LIN {X 0,Y 623.912,Z 1169.845,A -85,B 0,C 180,E1 30061.655,E2 30061.655} C_VEL
LIN {X 0,Y 623.911,Z 1170.404,A -85,B 0,C 180,E1 30059.543,E2 30059.543} C_VEL
LIN {X 0,Y 623.904,Z 1169.363,A -85,B 0,C 180,E1 30057.614,E2 30057.614} C_VEL
LIN {X 0,Y 623.916,Z 1166.7,A -85,B 0,C 180,E1 30055.682,E2 30055.682} C_VEL
LIN {X 0,Y 623.959,Z 1162.568,A -85,B 0,C 180,E1 30053.746,E2 30053.746} C_VEL
LIN {X 0,Y 624.049,Z 1156.994,A -85,B 0,C 180,E1 30051.897,E2 30051.897} C_VEL
LIN {X 0,Y 624.248,Z 1149.09,A -85,B 0,C 180,E1 30049.854,E2 30049.854} C_VEL
LIN {X 0,Y 624.565,Z 1140.192,A -85,B 0,C 180,E1 30047.99,E2 30047.99} C_VEL
LIN {X 0,Y 625.015,Z 1129.706,A -85,B 0,C 180,E1 30046.186,E2 30046.186} C_VEL
LIN {X 0,Y 625.63,Z 1117.625,A -85,B 0,C 180,E1 30044.427,E2 30044.427} C_VEL
LIN {X 0,Y 626.415,Z 1103.895,A -85,B 0,C 180,E1 30042.731,E2 30042.731} C_VEL
LIN {X 0,Y 627.334,Z 1088.573,A -85,B 0,C 180,E1 30041.124,E2 30041.124} C_VEL
LIN {X 0,Y 628.363,Z 1072.134,A -85,B 0,C 180,E1 30039.656,E2 30039.656} C_VEL
LIN {X 0,Y 629.487,Z 1054.056,A -85,B 0,C 180,E1 30038.281,E2 30038.281} C_VEL
LIN {X 0,Y 630.63,Z 1034.884,A -85,B 0,C 180,E1 30037.045,E2 30037.045} C_VEL
LIN {X 0,Y 631.734,Z 1015.659,A -85,B 0,C 180,E1 30036.001,E2 30036.001} C_VEL
LIN {X 0,Y 632.769,Z 994.956,A -85,B 0,C 180,E1 30035.077,E2 30035.077} C_VEL
LIN {X 0,Y 633.68,Z 974.386,A -85,B 0,C 180,E1 30034.336,E2 30034.336} C_VEL
LIN {X 0,Y 634.446,Z 952.859,A -85,B 0,C 180,E1 30033.726,E2 30033.726} C_VEL
LIN {X 0,Y 635.069,Z 931.038,A -85,B 0,C 180,E1 30033.278,E2 30033.278} C_VEL
LIN {X 0,Y 635.631,Z 892.123,A -85,B 0,C 180,E1 30032.768,E2 30032.768} C_VEL
LIN {X 0,Y 637.752,Z 731.192,A -85,B 0,C 180,E1 30030.768,E2 30030.768} C_VEL
LIN {X 0,Y 637.014,Z 723.617,A -85,B 0,C 180,E1 30030.63,E2 30030.63} C_VEL
LIN {X 0,Y 631.874,Z 703.847,A -85,B 0,C 180,E1 30030.101,E2 30030.101} C_VEL
LIN {X 0,Y 631.316,Z 697.339,A -85,B 0,C 180,E1 30029.982,E2 30029.982} C_VEL
LIN {X 0,Y 631.888,Z 655.219,A -85,B 0,C 180,E1 30029.42,E2 30029.42} C_VEL
LIN {X 0,Y 618.767,Z 628.94,A -85,B 0,C 180,E1 30028.33,E2 30028.33} C_VEL
LIN {X 0,Y 617.781,Z 626.772,A -85,B 0,C 180,E1 30028.226,E2 30028.226} C_VEL
LIN {X 0,Y 616.937,Z 623.823,A -85,B 0,C 180,E1 30027.835,E2 30027.835} C_VEL
LIN {X 0,Y 617.007,Z 623.813,A -85,B 0,C 180,E1 30024.762,E2 30024.762} C_VEL
LIN {X 0,Y 616.975,Z 623.812,A -85,B 0,C 180,E1 30021.636,E2 30021.636} C_VEL
LIN {X 0,Y 617.012,Z 623.805,A -85,B 0,C 180,E1 30018.478,E2 30018.478} C_VEL
LIN {X 0,Y 616.987,Z 623.813,A -85,B 0,C 180,E1 30015.221,E2 30015.221} C_VEL
LIN {X 0,Y 617.016,Z 623.81,A -85,B 0,C 180,E1 30012.085,E2 30012.085} C_VEL
LIN {X 0,Y 616.929,Z 623.818,A -85,B 0,C 180,E1 30009.078,E2 30009.078} C_VEL
LIN {X 0,Y 617.013,Z 623.809,A -85,B 0,C 180,E1 30006.034,E2 30006.034} C_VEL
LIN {X 0,Y 616.994,Z 623.814,A -85,B 0,C 180,E1 30002.882,E2 30002.882} C_VEL
LIN {X 0,Y 617.01,Z 623.806,A -85,B 0,C 180,E1 29999.622,E2 29999.622} C_VEL
LIN {X 0,Y 616.974,Z 623.811,A -85,B 0,C 180,E1 29996.551,E2 29996.551} C_VEL
LIN {X 0,Y 617.005,Z 623.814,A -85,B 0,C 180,E1 29993.394,E2 29993.394} C_VEL
LIN {X 0,Y 616.935,Z 623.817,A -85,B 0,C 180,E1 29990.394,E2 29990.394} C_VEL
LIN {X 0,Y 616.989,Z 623.809,A -85,B 0,C 180,E1 29987.253,E2 29987.253} C_VEL
LIN {X 0,Y 617.016,Z 623.808,A -85,B 0,C 180,E1 29984.165,E2 29984.165} C_VEL
LIN {X 0,Y 617.008,Z 623.81,A -85,B 0,C 180,E1 29980.889,E2 29980.889} C_VEL
LIN {X 0,Y 616.968,Z 623.808,A -85,B 0,C 180,E1 29977.825,E2 29977.825} C_VEL
LIN {X 0,Y 616.969,Z 623.815,A -85,B 0,C 180,E1 29974.697,E2 29974.697} C_VEL
LIN {X 0,Y 616.953,Z 623.81,A -85,B 0,C 180,E1 29971.673,E2 29971.673} C_VEL
LIN {X 0,Y 616.975,Z 623.81,A -85,B 0,C 180,E1 29968.515,E2 29968.515} C_VEL
LIN {X 0,Y 617.007,Z 623.807,A -85,B 0,C 180,E1 29965.447,E2 29965.447} C_VEL
LIN {X 0,Y 617.012,Z 623.811,A -85,B 0,C 180,E1 29962.271,E2 29962.271} C_VEL
LIN {X 0,Y 616.964,Z 623.804,A -85,B 0,C 180,E1 29959.26,E2 29959.26} C_VEL
LIN {X 0,Y 616.947,Z 623.816,A -85,B 0,C 180,E1 29956.027,E2 29956.027} C_VEL
LIN {X 0,Y 616.966,Z 623.815,A -85,B 0,C 180,E1 29953.138,E2 29953.138} C_VEL
LIN {X 0,Y 616.98,Z 623.809,A -85,B 0,C 180,E1 29950.006,E2 29950.006} C_VEL
LIN {X 0,Y 617.004,Z 623.809,A -85,B 0,C 180,E1 29946.912,E2 29946.912} C_VEL
LIN {X 0,Y 617.013,Z 623.812,A -85,B 0,C 180,E1 29943.744,E2 29943.744} C_VEL
LIN {X 0,Y 616.963,Z 623.813,A -85,B 0,C 180,E1 29940.698,E2 29940.698} C_VEL
LIN {X 0,Y 616.938,Z 623.817,A -85,B 0,C 180,E1 29937.429,E2 29937.429} C_VEL
LIN {X 0,Y 616.985,Z 623.816,A -85,B 0,C 180,E1 29934.539,E2 29934.539} C_VEL
LIN {X 0,Y 616.98,Z 623.811,A -85,B 0,C 180,E1 29931.36,E2 29931.36} C_VEL
LIN {X 0,Y 617,Z 623.81,A -85,B 0,C 180,E1 29928.334,E2 29928.334} C_VEL
LIN {X 0,Y 617.01,Z 623.811,A -85,B 0,C 180,E1 29925.179,E2 29925.179} C_VEL
LIN {X 0,Y 616.963,Z 623.816,A -85,B 0,C 180,E1 29922.137,E2 29922.137} C_VEL
LIN {X 0,Y 616.934,Z 623.827,A -85,B 0,C 180,E1 29920.696,E2 29920.696} C_VEL
LIN {X 0,Y 622.527,Z 645.232,A -85,B 0,C 180,E1 29918.834,E2 29918.834} C_VEL
LIN {X 0,Y 621.851,Z 690.99,A -85,B 0,C 180,E1 29915.395,E2 29915.395} C_VEL
LIN {X 0,Y 621.209,Z 730.49,A -85,B 0,C 180,E1 29912.408,E2 29912.408} C_VEL
LIN {X 0,Y 620.43,Z 772.737,A -85,B 0,C 180,E1 29909.227,E2 29909.227} C_VEL
LIN {X 0,Y 619.705,Z 815.192,A -85,B 0,C 180,E1 29906.029,E2 29906.029} C_VEL
LIN {X 0,Y 619.607,Z 824.743,A -85,B 0,C 180,E1 29905.342,E2 29905.342} C_VEL
LIN {X 0,Y 619.958,Z 832.218,A -85,B 0,C 180,E1 29905.238,E2 29905.238} C_VEL
LIN {X 0,Y 618.985,Z 967.136,A -85,B 0,C 180,E1 29903.544,E2 29903.544} C_VEL
LIN {X 0,Y 618.854,Z 983.402,A -85,B 0,C 180,E1 29903.165,E2 29903.165} C_VEL
LIN {X 0,Y 618.641,Z 999.258,A -85,B 0,C 180,E1 29902.621,E2 29902.621} C_VEL
LIN {X 0,Y 618.348,Z 1013.981,A -85,B 0,C 180,E1 29901.931,E2 29901.931} C_VEL
LIN {X 0,Y 618.043,Z 1027.886,A -85,B 0,C 180,E1 29901.096,E2 29901.096} C_VEL
LIN {X 0,Y 617.697,Z 1040.445,A -85,B 0,C 180,E1 29900.144,E2 29900.144} C_VEL
LIN {X 0,Y 617.356,Z 1052.594,A -85,B 0,C 180,E1 29898.996,E2 29898.996} C_VEL
LIN {X 0,Y 617.064,Z 1062.411,A -85,B 0,C 180,E1 29897.831,E2 29897.831} C_VEL
LIN {X 0,Y 616.819,Z 1071.471,A -85,B 0,C 180,E1 29896.478,E2 29896.478} C_VEL
LIN {X 0,Y 616.646,Z 1078.364,A -85,B 0,C 180,E1 29895.131,E2 29895.131} C_VEL
LIN {X 0,Y 616.54,Z 1083.784,A -85,B 0,C 180,E1 29893.694,E2 29893.694} C_VEL
LIN {X 0,Y 616.468,Z 1087.777,A -85,B 0,C 180,E1 29892.039,E2 29892.039} C_VEL
LIN {X 0,Y 616.45,Z 1089.511,A -85,B 0,C 180,E1 29890.559,E2 29890.559} C_VEL
LIN {X 0,Y 616.474,Z 1089.436,A -85,B 0,C 180,E1 29889.05,E2 29889.05} C_VEL
LIN {X 0,Y 616.534,Z 1087.628,A -85,B 0,C 180,E1 29887.546,E2 29887.546} C_VEL
LIN {X 0,Y 616.626,Z 1083.923,A -85,B 0,C 180,E1 29886.048,E2 29886.048} C_VEL
LIN {X 0,Y 616.778,Z 1078.713,A -85,B 0,C 180,E1 29884.647,E2 29884.647} C_VEL
LIN {X 0,Y 616.991,Z 1071.524,A -85,B 0,C 180,E1 29883.25,E2 29883.25} C_VEL
LIN {X 0,Y 617.267,Z 1062.829,A -85,B 0,C 180,E1 29881.947,E2 29881.947} C_VEL
LIN {X 0,Y 617.594,Z 1052.516,A -85,B 0,C 180,E1 29880.74,E2 29880.74} C_VEL
LIN {X 0,Y 617.96,Z 1040.631,A -85,B 0,C 180,E1 29879.627,E2 29879.627} C_VEL
LIN {X 0,Y 618.306,Z 1027.459,A -85,B 0,C 180,E1 29878.654,E2 29878.654} C_VEL
LIN {X 0,Y 618.576,Z 1014.097,A -85,B 0,C 180,E1 29877.867,E2 29877.867} C_VEL
LIN {X 0,Y 618.83,Z 999.677,A -85,B 0,C 180,E1 29877.22,E2 29877.22} C_VEL
LIN {X 0,Y 619.005,Z 985.719,A -85,B 0,C 180,E1 29876.748,E2 29876.748} C_VEL
LIN {X 0,Y 619.098,Z 970.478,A -85,B 0,C 180,E1 29876.378,E2 29876.378} C_VEL
LIN {X 0,Y 619.279,Z 928.275,A -85,B 0,C 180,E1 29875.826,E2 29875.826} C_VEL
LIN {X 0,Y 620.272,Z 827.99,A -85,B 0,C 180,E1 29874.517,E2 29874.517} C_VEL
LIN {X 0,Y 620.921,Z 785.093,A -85,B 0,C 180,E1 29871.338,E2 29871.338} C_VEL
LIN {X 0,Y 621.362,Z 749.405,A -85,B 0,C 180,E1 29868.723,E2 29868.723} C_VEL
LIN {X 0,Y 621.787,Z 707.503,A -85,B 0,C 180,E1 29865.708,E2 29865.708} C_VEL
LIN {X 0,Y 621.849,Z 662.544,A -85,B 0,C 180,E1 29862.548,E2 29862.548} C_VEL
LIN {X 0,Y 621.705,Z 640.309,A -85,B 0,C 180,E1 29861.022,E2 29861.022} C_VEL
LIN {X 0,Y 616.991,Z 623.817,A -85,B 0,C 180,E1 29859.681,E2 29859.681} C_VEL
LIN {X 0,Y 616.981,Z 623.82,A -85,B 0,C 180,E1 29856.706,E2 29856.706} C_VEL
LIN {X 0,Y 617.01,Z 623.814,A -85,B 0,C 180,E1 29853.326,E2 29853.326} C_VEL
LIN {X 0,Y 617.018,Z 623.814,A -85,B 0,C 180,E1 29850.105,E2 29850.105} C_VEL
LIN {X 0,Y 616.973,Z 623.815,A -85,B 0,C 180,E1 29846.895,E2 29846.895} C_VEL
LIN {X 0,Y 616.987,Z 623.814,A -85,B 0,C 180,E1 29843.963,E2 29843.963} C_VEL
LIN {X 0,Y 617.01,Z 623.814,A -85,B 0,C 180,E1 29840.68,E2 29840.68} C_VEL
LIN {X 0,Y 617.019,Z 623.81,A -85,B 0,C 180,E1 29837.486,E2 29837.486} C_VEL
LIN {X 0,Y 616.973,Z 623.813,A -85,B 0,C 180,E1 29834.247,E2 29834.247} C_VEL
LIN {X 0,Y 617.021,Z 623.809,A -85,B 0,C 180,E1 29831.016,E2 29831.016} C_VEL
LIN {X 0,Y 617.006,Z 623.811,A -85,B 0,C 180,E1 29827.887,E2 29827.887} C_VEL
LIN {X 0,Y 617.049,Z 624.04,A -85,B 0,C 180,E1 29826.952,E2 29826.952} C_VEL
LIN {X 0,Y 624.996,Z 648.862,A -85,B 0,C 180,E1 29824.16,E2 29824.16} C_VEL
LIN {X 0,Y 627.248,Z 656.87,A -85,B 0,C 180,E1 29823.308,E2 29823.308} C_VEL
LIN {X 0,Y 626.069,Z 680.989,A -85,B 0,C 180,E1 29821.26,E2 29821.26} C_VEL
LIN {X 0,Y 631.821,Z 709.359,A -85,B 0,C 180,E1 29820.55,E2 29820.55} C_VEL
LIN {X 0,Y 628.74,Z 911.351,A -85,B 0,C 180,E1 29817.97,E2 29817.97} C_VEL
LIN {X 0,Y 627.625,Z 986.56,A -85,B 0,C 180,E1 29816.998,E2 29816.998} C_VEL
LIN {X 0,Y 626.902,Z 1008.567,A -85,B 0,C 180,E1 29816.549,E2 29816.549} C_VEL
LIN {X 0,Y 626.04,Z 1030.132,A -85,B 0,C 180,E1 29815.944,E2 29815.944} C_VEL
LIN {X 0,Y 625.036,Z 1051.381,A -85,B 0,C 180,E1 29815.182,E2 29815.182} C_VEL
LIN {X 0,Y 623.929,Z 1072.004,A -85,B 0,C 180,E1 29814.265,E2 29814.265} C_VEL
LIN {X 0,Y 622.789,Z 1091.493,A -85,B 0,C 180,E1 29813.212,E2 29813.212} C_VEL
LIN {X 0,Y 621.585,Z 1111.078,A -85,B 0,C 180,E1 29811.961,E2 29811.961} C_VEL
LIN {X 0,Y 620.498,Z 1128.452,A -85,B 0,C 180,E1 29810.663,E2 29810.663} C_VEL
LIN {X 0,Y 619.474,Z 1144.894,A -85,B 0,C 180,E1 29809.22,E2 29809.22} C_VEL
LIN {X 0,Y 618.568,Z 1159.94,A -85,B 0,C 180,E1 29807.69,E2 29807.69} C_VEL
LIN {X 0,Y 617.799,Z 1173.773,A -85,B 0,C 180,E1 29806.065,E2 29806.065} C_VEL
LIN {X 0,Y 617.156,Z 1186.266,A -85,B 0,C 180,E1 29804.334,E2 29804.334} C_VEL
LIN {X 0,Y 616.677,Z 1197.217,A -85,B 0,C 180,E1 29802.547,E2 29802.547} C_VEL
LIN {X 0,Y 616.353,Z 1206.523,A -85,B 0,C 180,E1 29800.751,E2 29800.751} C_VEL
LIN {X 0,Y 616.121,Z 1214.386,A -85,B 0,C 180,E1 29798.867,E2 29798.867} C_VEL
LIN {X 0,Y 615.98,Z 1220.89,A -85,B 0,C 180,E1 29796.898,E2 29796.898} C_VEL
LIN {X 0,Y 615.92,Z 1225.641,A -85,B 0,C 180,E1 29794.935,E2 29794.935} C_VEL
LIN {X 0,Y 615.904,Z 1228.673,A -85,B 0,C 180,E1 29792.977,E2 29792.977} C_VEL
LIN {X 0,Y 615.91,Z 1230.28,A -85,B 0,C 180,E1 29790.929,E2 29790.929} C_VEL
LIN {X 0,Y 615.91,Z 1230.279,A -85,B 0,C 180,E1 29789.069,E2 29789.069} C_VEL
LIN {X 0,Y 615.905,Z 1228.666,A -85,B 0,C 180,E1 29787.021,E2 29787.021} C_VEL
LIN {X 0,Y 615.92,Z 1225.63,A -85,B 0,C 180,E1 29785.063,E2 29785.063} C_VEL
LIN {X 0,Y 615.981,Z 1220.882,A -85,B 0,C 180,E1 29783.1,E2 29783.1} C_VEL
LIN {X 0,Y 616.119,Z 1214.356,A -85,B 0,C 180,E1 29781.13,E2 29781.13} C_VEL
LIN {X 0,Y 616.35,Z 1206.432,A -85,B 0,C 180,E1 29779.247,E2 29779.247} C_VEL
LIN {X 0,Y 616.699,Z 1196.523,A -85,B 0,C 180,E1 29777.355,E2 29777.355} C_VEL
LIN {X 0,Y 617.182,Z 1185.19,A -85,B 0,C 180,E1 29775.551,E2 29775.551} C_VEL
LIN {X 0,Y 617.807,Z 1172.49,A -85,B 0,C 180,E1 29773.836,E2 29773.836} C_VEL
LIN {X 0,Y 618.569,Z 1158.134,A -85,B 0,C 180,E1 29772.196,E2 29772.196} C_VEL
LIN {X 0,Y 619.47,Z 1142.089,A -85,B 0,C 180,E1 29770.627,E2 29770.627} C_VEL
LIN {X 0,Y 620.503,Z 1124.219,A -85,B 0,C 180,E1 29769.137,E2 29769.137} C_VEL
LIN {X 0,Y 621.53,Z 1105.923,A -85,B 0,C 180,E1 29767.835,E2 29767.835} C_VEL
LIN {X 0,Y 622.596,Z 1086.571,A -85,B 0,C 180,E1 29766.678,E2 29766.678} C_VEL
LIN {X 0,Y 623.608,Z 1066.417,A -85,B 0,C 180,E1 29765.664,E2 29765.664} C_VEL
LIN {X 0,Y 624.581,Z 1045.558,A -85,B 0,C 180,E1 29764.795,E2 29764.795} C_VEL
LIN {X 0,Y 625.479,Z 1023.937,A -85,B 0,C 180,E1 29764.073,E2 29764.073} C_VEL
LIN {X 0,Y 626.217,Z 1002.185,A -85,B 0,C 180,E1 29763.519,E2 29763.519} C_VEL
LIN {X 0,Y 626.845,Z 978.254,A -85,B 0,C 180,E1 29763.087,E2 29763.087} C_VEL
LIN {X 0,Y 628.923,Z 830.62,A -85,B 0,C 180,E1 29761.18,E2 29761.18} C_VEL
LIN {X 0,Y 631.767,Z 708.547,A -85,B 0,C 180,E1 29759.452,E2 29759.452} C_VEL
LIN {X 0,Y 625.568,Z 675.462,A -85,B 0,C 180,E1 29758.5,E2 29758.5} C_VEL
LIN {X 0,Y 626.748,Z 655.477,A -85,B 0,C 180,E1 29756.714,E2 29756.714} C_VEL
LIN {X 0,Y 622.75,Z 640.651,A -85,B 0,C 180,E1 29754.972,E2 29754.972} C_VEL
LIN {X 0,Y 619,Z 629.633,A -85,B 0,C 180,E1 29753.487,E2 29753.487} C_VEL
LIN {X 0,Y 617.009,Z 623.813,A -85,B 0,C 180,E1 29752.602,E2 29752.602} C_VEL
LIN {X 0,Y 616.98,Z 623.818,A -85,B 0,C 180,E1 29749.59,E2 29749.59} C_VEL
LIN {X 0,Y 617.013,Z 623.813,A -85,B 0,C 180,E1 29746.47,E2 29746.47} C_VEL
LIN {X 0,Y 616.971,Z 623.817,A -85,B 0,C 180,E1 29743.407,E2 29743.407} C_VEL
LIN {X 0,Y 617.018,Z 623.813,A -85,B 0,C 180,E1 29740.286,E2 29740.286} C_VEL
LIN {X 0,Y 616.963,Z 623.817,A -85,B 0,C 180,E1 29737.273,E2 29737.273} C_VEL
LIN {X 0,Y 617.019,Z 623.812,A -85,B 0,C 180,E1 29734.218,E2 29734.218} C_VEL
LIN {X 0,Y 616.979,Z 623.96,A -85,B 0,C 180,E1 29733.382,E2 29733.382} C_VEL
LIN {X 0,Y 620.268,Z 633.467,A -85,B 0,C 180,E1 29731.798,E2 29731.798} C_VEL
LIN {X 0,Y 628.034,Z 646.969,A -85,B 0,C 180,E1 29731.002,E2 29731.002} C_VEL
LIN {X 0,Y 632.541,Z 656.333,A -85,B 0,C 180,E1 29730.544,E2 29730.544} C_VEL
LIN {X 0,Y 629.48,Z 777.376,A -85,B 0,C 180,E1 29728.801,E2 29728.801} C_VEL
LIN {X 0,Y 627.398,Z 908.624,A -85,B 0,C 180,E1 29727.084,E2 29727.084} C_VEL
LIN {X 0,Y 626.891,Z 937.237,A -85,B 0,C 180,E1 29726.668,E2 29726.668} C_VEL
LIN {X 0,Y 626.321,Z 959.429,A -85,B 0,C 180,E1 29726.177,E2 29726.177} C_VEL
LIN {X 0,Y 625.546,Z 980.68,A -85,B 0,C 180,E1 29725.544,E2 29725.544} C_VEL
LIN {X 0,Y 624.643,Z 1001.442,A -85,B 0,C 180,E1 29724.747,E2 29724.747} C_VEL
LIN {X 0,Y 623.606,Z 1021.962,A -85,B 0,C 180,E1 29723.783,E2 29723.783} C_VEL
LIN {X 0,Y 622.581,Z 1040.772,A -85,B 0,C 180,E1 29722.723,E2 29722.723} C_VEL
LIN {X 0,Y 621.481,Z 1058.677,A -85,B 0,C 180,E1 29721.522,E2 29721.522} C_VEL
LIN {X 0,Y 620.415,Z 1075.722,A -85,B 0,C 180,E1 29720.177,E2 29720.177} C_VEL
LIN {X 0,Y 619.416,Z 1091.38,A -85,B 0,C 180,E1 29718.739,E2 29718.739} C_VEL
LIN {X 0,Y 618.483,Z 1106.471,A -85,B 0,C 180,E1 29717.113,E2 29717.113} C_VEL
LIN {X 0,Y 617.681,Z 1119.911,A -85,B 0,C 180,E1 29715.397,E2 29715.397} C_VEL
LIN {X 0,Y 617.043,Z 1131.871,A -85,B 0,C 180,E1 29713.591,E2 29713.591} C_VEL
LIN {X 0,Y 616.563,Z 1142.344,A -85,B 0,C 180,E1 29711.698,E2 29711.698} C_VEL
LIN {X 0,Y 616.255,Z 1150.933,A -85,B 0,C 180,E1 29709.811,E2 29709.811} C_VEL
LIN {X 0,Y 616.053,Z 1158.018,A -85,B 0,C 180,E1 29707.838,E2 29707.838} C_VEL
LIN {X 0,Y 615.948,Z 1163.903,A -85,B 0,C 180,E1 29705.669,E2 29705.669} C_VEL
LIN {X 0,Y 615.915,Z 1167.665,A -85,B 0,C 180,E1 29703.725,E2 29703.725} C_VEL
LIN {X 0,Y 615.91,Z 1169.775,A -85,B 0,C 180,E1 29701.77,E2 29701.77} C_VEL
LIN {X 0,Y 615.905,Z 1170.449,A -85,B 0,C 180,E1 29699.723,E2 29699.723} C_VEL
LIN {X 0,Y 615.902,Z 1169.569,A -85,B 0,C 180,E1 29697.862,E2 29697.862} C_VEL
LIN {X 0,Y 615.91,Z 1167.023,A -85,B 0,C 180,E1 29695.813,E2 29695.813} C_VEL
LIN {X 0,Y 615.947,Z 1163.241,A -85,B 0,C 180,E1 29693.945,E2 29693.945} C_VEL
LIN {X 0,Y 616.051,Z 1157.696,A -85,B 0,C 180,E1 29691.978,E2 29691.978} C_VEL
LIN {X 0,Y 616.26,Z 1150.491,A -85,B 0,C 180,E1 29690.005,E2 29690.005} C_VEL
LIN {X 0,Y 616.58,Z 1141.807,A -85,B 0,C 180,E1 29688.117,E2 29688.117} C_VEL
LIN {X 0,Y 617.064,Z 1131.192,A -85,B 0,C 180,E1 29686.222,E2 29686.222} C_VEL
LIN {X 0,Y 617.723,Z 1118.936,A -85,B 0,C 180,E1 29684.39,E2 29684.39} C_VEL
LIN {X 0,Y 618.531,Z 1105.593,A -85,B 0,C 180,E1 29682.698,E2 29682.698} C_VEL
LIN {X 0,Y 619.497,Z 1090.283,A -85,B 0,C 180,E1 29681.055,E2 29681.055} C_VEL
LIN {X 0,Y 620.598,Z 1073.703,A -85,B 0,C 180,E1 29679.538,E2 29679.538} C_VEL
LIN {X 0,Y 621.774,Z 1055.841,A -85,B 0,C 180,E1 29678.146,E2 29678.146} C_VEL
LIN {X 0,Y 622.937,Z 1037.8,A -85,B 0,C 180,E1 29676.946,E2 29676.946} C_VEL
LIN {X 0,Y 624.116,Z 1018.173,A -85,B 0,C 180,E1 29675.849,E2 29675.849} C_VEL
LIN {X 0,Y 625.187,Z 998.226,A -85,B 0,C 180,E1 29674.926,E2 29674.926} C_VEL
LIN {X 0,Y 626.198,Z 977.222,A -85,B 0,C 180,E1 29674.134,E2 29674.134} C_VEL
LIN {X 0,Y 627.058,Z 955.646,A -85,B 0,C 180,E1 29673.494,E2 29673.494} C_VEL
LIN {X 0,Y 627.691,Z 933.727,A -85,B 0,C 180,E1 29673.025,E2 29673.025} C_VEL
LIN {X 0,Y 628.228,Z 904.066,A -85,B 0,C 180,E1 29672.608,E2 29672.608} C_VEL
LIN {X 0,Y 631.316,Z 697.339,A -85,B 0,C 180,E1 29669.982,E2 29669.982} C_VEL
LIN {X 0,Y 630.577,Z 689.773,A -85,B 0,C 180,E1 29669.838,E2 29669.838} C_VEL
LIN {X 0,Y 625.54,Z 670.016,A -85,B 0,C 180,E1 29669.294,E2 29669.294} C_VEL
LIN {X 0,Y 624.995,Z 663.512,A -85,B 0,C 180,E1 29669.173,E2 29669.173} C_VEL
LIN {X 0,Y 624.879,Z 657.552,A -85,B 0,C 180,E1 29669.081,E2 29669.081} C_VEL
LIN {X 0,Y 611.174,Z 630.338,A -85,B 0,C 180,E1 29667.915,E2 29667.915} C_VEL
LIN {X 0,Y 609.654,Z 627.14,A -85,B 0,C 180,E1 29667.767,E2 29667.767} C_VEL
LIN {X 0,Y 608.993,Z 624.813,A -85,B 0,C 180,E1 29667.447,E2 29667.447} C_VEL
LIN {X 0,Y 609.041,Z 624.803,A -85,B 0,C 180,E1 29664.239,E2 29664.239} C_VEL
LIN {X 0,Y 609.069,Z 624.803,A -85,B 0,C 180,E1 29661.166,E2 29661.166} C_VEL
LIN {X 0,Y 609.062,Z 624.797,A -85,B 0,C 180,E1 29657.907,E2 29657.907} C_VEL
LIN {X 0,Y 609.038,Z 624.8,A -85,B 0,C 180,E1 29654.831,E2 29654.831} C_VEL
LIN {X 0,Y 609.043,Z 624.806,A -85,B 0,C 180,E1 29651.674,E2 29651.674} C_VEL
LIN {X 0,Y 609.004,Z 624.807,A -85,B 0,C 180,E1 29648.723,E2 29648.723} C_VEL
LIN {X 0,Y 609.029,Z 624.799,A -85,B 0,C 180,E1 29645.485,E2 29645.485} C_VEL
LIN {X 0,Y 609.074,Z 624.8,A -85,B 0,C 180,E1 29642.461,E2 29642.461} C_VEL
LIN {X 0,Y 609.068,Z 624.799,A -85,B 0,C 180,E1 29639.29,E2 29639.29} C_VEL
LIN {X 0,Y 609.038,Z 624.798,A -85,B 0,C 180,E1 29636.209,E2 29636.209} C_VEL
LIN {X 0,Y 609.01,Z 624.803,A -85,B 0,C 180,E1 29632.926,E2 29632.926} C_VEL
LIN {X 0,Y 609.032,Z 624.806,A -85,B 0,C 180,E1 29629.969,E2 29629.969} C_VEL
LIN {X 0,Y 609.028,Z 624.8,A -85,B 0,C 180,E1 29626.796,E2 29626.796} C_VEL
LIN {X 0,Y 609.067,Z 624.793,A -85,B 0,C 180,E1 29623.772,E2 29623.772} C_VEL
LIN {X 0,Y 609.07,Z 624.803,A -85,B 0,C 180,E1 29620.501,E2 29620.501} C_VEL
LIN {X 0,Y 609.056,Z 624.795,A -85,B 0,C 180,E1 29617.358,E2 29617.358} C_VEL
LIN {X 0,Y 608.994,Z 624.803,A -85,B 0,C 180,E1 29614.238,E2 29614.238} C_VEL
LIN {X 0,Y 609.076,Z 624.801,A -85,B 0,C 180,E1 29611.13,E2 29611.13} C_VEL
LIN {X 0,Y 609.036,Z 624.801,A -85,B 0,C 180,E1 29608.026,E2 29608.026} C_VEL
LIN {X 0,Y 609.072,Z 624.79,A -85,B 0,C 180,E1 29604.821,E2 29604.821} C_VEL
LIN {X 0,Y 609.044,Z 624.799,A -85,B 0,C 180,E1 29601.6,E2 29601.6} C_VEL
LIN {X 0,Y 609.074,Z 624.791,A -85,B 0,C 180,E1 29598.448,E2 29598.448} C_VEL
LIN {X 0,Y 608.989,Z 624.805,A -85,B 0,C 180,E1 29595.453,E2 29595.453} C_VEL
LIN {X 0,Y 609.05,Z 624.799,A -85,B 0,C 180,E1 29592.321,E2 29592.321} C_VEL
LIN {X 0,Y 609.064,Z 624.802,A -85,B 0,C 180,E1 29589.233,E2 29589.233} C_VEL
LIN {X 0,Y 609.066,Z 624.796,A -85,B 0,C 180,E1 29585.977,E2 29585.977} C_VEL
LIN {X 0,Y 609.038,Z 624.8,A -85,B 0,C 180,E1 29582.952,E2 29582.952} C_VEL
LIN {X 0,Y 609.062,Z 624.804,A -85,B 0,C 180,E1 29579.846,E2 29579.846} C_VEL
LIN {X 0,Y 608.997,Z 624.806,A -85,B 0,C 180,E1 29576.856,E2 29576.856} C_VEL
LIN {X 0,Y 609.033,Z 624.8,A -85,B 0,C 180,E1 29573.553,E2 29573.553} C_VEL
LIN {X 0,Y 609.074,Z 624.802,A -85,B 0,C 180,E1 29570.491,E2 29570.491} C_VEL
LIN {X 0,Y 609.068,Z 624.8,A -85,B 0,C 180,E1 29567.314,E2 29567.314} C_VEL
LIN {X 0,Y 609.036,Z 624.802,A -85,B 0,C 180,E1 29564.242,E2 29564.242} C_VEL
LIN {X 0,Y 609.015,Z 624.843,A -85,B 0,C 180,E1 29560.957,E2 29560.957} C_VEL
LIN {X 0,Y 614.93,Z 647.129,A -85,B 0,C 180,E1 29558.993,E2 29558.993} C_VEL
LIN {X 0,Y 614.222,Z 691.425,A -85,B 0,C 180,E1 29555.643,E2 29555.643} C_VEL
LIN {X 0,Y 613.557,Z 731.688,A -85,B 0,C 180,E1 29552.595,E2 29552.595} C_VEL
LIN {X 0,Y 612.717,Z 774.101,A -85,B 0,C 180,E1 29549.379,E2 29549.379} C_VEL
LIN {X 0,Y 611.96,Z 816.445,A -85,B 0,C 180,E1 29546.175,E2 29546.175} C_VEL
LIN {X 0,Y 611.854,Z 825.417,A -85,B 0,C 180,E1 29545.524,E2 29545.524} C_VEL
LIN {X 0,Y 612.206,Z 832.974,A -85,B 0,C 180,E1 29545.416,E2 29545.416} C_VEL
LIN {X 0,Y 611.162,Z 968.04,A -85,B 0,C 180,E1 29543.688,E2 29543.688} C_VEL
LIN {X 0,Y 611.028,Z 984.393,A -85,B 0,C 180,E1 29543.3,E2 29543.3} C_VEL
LIN {X 0,Y 610.815,Z 999.568,A -85,B 0,C 180,E1 29542.774,E2 29542.774} C_VEL
LIN {X 0,Y 610.511,Z 1014.46,A -85,B 0,C 180,E1 29542.076,E2 29542.076} C_VEL
LIN {X 0,Y 610.177,Z 1029.016,A -85,B 0,C 180,E1 29541.192,E2 29541.192} C_VEL
LIN {X 0,Y 609.805,Z 1041.758,A -85,B 0,C 180,E1 29540.208,E2 29540.208} C_VEL
LIN {X 0,Y 609.454,Z 1053.779,A -85,B 0,C 180,E1 29539.053,E2 29539.053} C_VEL
LIN {X 0,Y 609.123,Z 1064.262,A -85,B 0,C 180,E1 29537.775,E2 29537.775} C_VEL
LIN {X 0,Y 608.884,Z 1072.789,A -85,B 0,C 180,E1 29536.466,E2 29536.466} C_VEL
LIN {X 0,Y 608.695,Z 1079.955,A -85,B 0,C 180,E1 29535.016,E2 29535.016} C_VEL
LIN {X 0,Y 608.594,Z 1085.137,A -85,B 0,C 180,E1 29533.586,E2 29533.586} C_VEL
LIN {X 0,Y 608.519,Z 1088.89,A -85,B 0,C 180,E1 29531.946,E2 29531.946} C_VEL
LIN {X 0,Y 608.505,Z 1090.475,A -85,B 0,C 180,E1 29530.507,E2 29530.507} C_VEL
LIN {X 0,Y 608.535,Z 1090.359,A -85,B 0,C 180,E1 29528.978,E2 29528.978} C_VEL
LIN {X 0,Y 608.602,Z 1088.497,A -85,B 0,C 180,E1 29527.455,E2 29527.455} C_VEL
LIN {X 0,Y 608.709,Z 1084.728,A -85,B 0,C 180,E1 29525.938,E2 29525.938} C_VEL
LIN {X 0,Y 608.881,Z 1079.447,A -85,B 0,C 180,E1 29524.519,E2 29524.519} C_VEL
LIN {X 0,Y 609.115,Z 1072.156,A -85,B 0,C 180,E1 29523.103,E2 29523.103} C_VEL
LIN {X 0,Y 609.415,Z 1063.348,A -85,B 0,C 180,E1 29521.784,E2 29521.784} C_VEL
LIN {X 0,Y 609.771,Z 1052.896,A -85,B 0,C 180,E1 29520.562,E2 29520.562} C_VEL
LIN {X 0,Y 610.146,Z 1041.389,A -85,B 0,C 180,E1 29519.482,E2 29519.482} C_VEL
LIN {X 0,Y 610.516,Z 1028.178,A -85,B 0,C 180,E1 29518.496,E2 29518.496} C_VEL
LIN {X 0,Y 610.807,Z 1014.75,A -85,B 0,C 180,E1 29517.699,E2 29517.699} C_VEL
LIN {X 0,Y 611.073,Z 1000.207,A -85,B 0,C 180,E1 29517.044,E2 29517.044} C_VEL
LIN {X 0,Y 611.253,Z 986.753,A -85,B 0,C 180,E1 29516.584,E2 29516.584} C_VEL
LIN {X 0,Y 611.352,Z 971.731,A -85,B 0,C 180,E1 29516.212,E2 29516.212} C_VEL
LIN {X 0,Y 611.505,Z 934.063,A -85,B 0,C 180,E1 29515.706,E2 29515.706} C_VEL
LIN {X 0,Y 612.651,Z 829.039,A -85,B 0,C 180,E1 29514.308,E2 29514.308} C_VEL
LIN {X 0,Y 613.342,Z 787.124,A -85,B 0,C 180,E1 29511.183,E2 29511.183} C_VEL
LIN {X 0,Y 613.883,Z 747.218,A -85,B 0,C 180,E1 29508.251,E2 29508.251} C_VEL
LIN {X 0,Y 614.266,Z 706.057,A -85,B 0,C 180,E1 29505.288,E2 29505.288} C_VEL
LIN {X 0,Y 614.33,Z 669.711,A -85,B 0,C 180,E1 29502.718,E2 29502.718} C_VEL
LIN {X 0,Y 614.306,Z 642.831,A -85,B 0,C 180,E1 29500.852,E2 29500.852} C_VEL
LIN {X 0,Y 609.036,Z 624.807,A -85,B 0,C 180,E1 29499.352,E2 29499.352} C_VEL
LIN {X 0,Y 609.038,Z 624.809,A -85,B 0,C 180,E1 29496.486,E2 29496.486} C_VEL
LIN {X 0,Y 609.073,Z 624.805,A -85,B 0,C 180,E1 29493.161,E2 29493.161} C_VEL
LIN {X 0,Y 609.081,Z 624.801,A -85,B 0,C 180,E1 29489.895,E2 29489.895} C_VEL
LIN {X 0,Y 609.033,Z 624.805,A -85,B 0,C 180,E1 29486.632,E2 29486.632} C_VEL
LIN {X 0,Y 609.069,Z 624.801,A -85,B 0,C 180,E1 29483.537,E2 29483.537} C_VEL
LIN {X 0,Y 609.065,Z 624.802,A -85,B 0,C 180,E1 29480.346,E2 29480.346} C_VEL
LIN {X 0,Y 609.067,Z 624.799,A -85,B 0,C 180,E1 29477.053,E2 29477.053} C_VEL
LIN {X 0,Y 609.05,Z 624.802,A -85,B 0,C 180,E1 29473.885,E2 29473.885} C_VEL
LIN {X 0,Y 609.071,Z 624.798,A -85,B 0,C 180,E1 29470.795,E2 29470.795} C_VEL
LIN {X 0,Y 609.059,Z 624.799,A -85,B 0,C 180,E1 29467.639,E2 29467.639} C_VEL
LIN {X 0,Y 609.07,Z 624.876,A -85,B 0,C 180,E1 29467.384,E2 29467.384} C_VEL
LIN {X 0,Y 617.292,Z 650.469,A -85,B 0,C 180,E1 29464.463,E2 29464.463} C_VEL
LIN {X 0,Y 619.881,Z 659.545,A -85,B 0,C 180,E1 29463.479,E2 29463.479} C_VEL
LIN {X 0,Y 618.776,Z 680.643,A -85,B 0,C 180,E1 29461.664,E2 29461.664} C_VEL
LIN {X 0,Y 624.871,Z 710.814,A -85,B 0,C 180,E1 29460.898,E2 29460.898} C_VEL
LIN {X 0,Y 621.006,Z 946.426,A -85,B 0,C 180,E1 29457.838,E2 29457.838} C_VEL
LIN {X 0,Y 620.288,Z 987.493,A -85,B 0,C 180,E1 29457.282,E2 29457.282} C_VEL
LIN {X 0,Y 619.525,Z 1009.238,A -85,B 0,C 180,E1 29456.827,E2 29456.827} C_VEL
LIN {X 0,Y 618.615,Z 1030.294,A -85,B 0,C 180,E1 29456.223,E2 29456.223} C_VEL
LIN {X 0,Y 617.56,Z 1051.314,A -85,B 0,C 180,E1 29455.457,E2 29455.457} C_VEL
LIN {X 0,Y 616.357,Z 1072.425,A -85,B 0,C 180,E1 29454.504,E2 29454.504} C_VEL
LIN {X 0,Y 615.127,Z 1092.175,A -85,B 0,C 180,E1 29453.416,E2 29453.416} C_VEL
LIN {X 0,Y 613.853,Z 1111.57,A -85,B 0,C 180,E1 29452.151,E2 29452.151} C_VEL
LIN {X 0,Y 612.667,Z 1129.375,A -85,B 0,C 180,E1 29450.79,E2 29450.79} C_VEL
LIN {X 0,Y 611.573,Z 1146.209,A -85,B 0,C 180,E1 29449.283,E2 29449.283} C_VEL
LIN {X 0,Y 610.625,Z 1161.009,A -85,B 0,C 180,E1 29447.731,E2 29447.731} C_VEL
LIN {X 0,Y 609.788,Z 1175.326,A -85,B 0,C 180,E1 29445.989,E2 29445.989} C_VEL
LIN {X 0,Y 609.141,Z 1187.546,A -85,B 0,C 180,E1 29444.252,E2 29444.252} C_VEL
LIN {X 0,Y 608.649,Z 1198.281,A -85,B 0,C 180,E1 29442.426,E2 29442.426} C_VEL
LIN {X 0,Y 608.292,Z 1208.126,A -85,B 0,C 180,E1 29440.416,E2 29440.416} C_VEL
LIN {X 0,Y 608.102,Z 1215.718,A -85,B 0,C 180,E1 29438.509,E2 29438.509} C_VEL
LIN {X 0,Y 607.974,Z 1221.543,A -85,B 0,C 180,E1 29436.602,E2 29436.602} C_VEL
LIN {X 0,Y 607.928,Z 1226.197,A -85,B 0,C 180,E1 29434.527,E2 29434.527} C_VEL
LIN {X 0,Y 607.914,Z 1229.041,A -85,B 0,C 180,E1 29432.544,E2 29432.544} C_VEL
LIN {X 0,Y 607.903,Z 1230.2,A -85,B 0,C 180,E1 29430.564,E2 29430.564} C_VEL
LIN {X 0,Y 607.9,Z 1229.899,A -85,B 0,C 180,E1 29428.585,E2 29428.585} C_VEL
LIN {X 0,Y 607.907,Z 1228.094,A -85,B 0,C 180,E1 29426.699,E2 29426.699} C_VEL
LIN {X 0,Y 607.94,Z 1224.465,A -85,B 0,C 180,E1 29424.619,E2 29424.619} C_VEL
LIN {X 0,Y 608.018,Z 1219.359,A -85,B 0,C 180,E1 29422.629,E2 29422.629} C_VEL
LIN {X 0,Y 608.165,Z 1212.366,A -85,B 0,C 180,E1 29420.631,E2 29420.631} C_VEL
LIN {X 0,Y 608.434,Z 1203.471,A -85,B 0,C 180,E1 29418.625,E2 29418.625} C_VEL
LIN {X 0,Y 608.829,Z 1193.646,A -85,B 0,C 180,E1 29416.803,E2 29416.803} C_VEL
LIN {X 0,Y 609.379,Z 1181.761,A -85,B 0,C 180,E1 29414.973,E2 29414.973} C_VEL
LIN {X 0,Y 610.078,Z 1168.398,A -85,B 0,C 180,E1 29413.233,E2 29413.233} C_VEL
LIN {X 0,Y 610.959,Z 1153.09,A -85,B 0,C 180,E1 29411.537,E2 29411.537} C_VEL
LIN {X 0,Y 611.932,Z 1136.606,A -85,B 0,C 180,E1 29409.978,E2 29409.978} C_VEL
LIN {X 0,Y 612.978,Z 1119.013,A -85,B 0,C 180,E1 29408.568,E2 29408.568} C_VEL
LIN {X 0,Y 614.078,Z 1100.498,A -85,B 0,C 180,E1 29407.299,E2 29407.299} C_VEL
LIN {X 0,Y 615.167,Z 1081.238,A -85,B 0,C 180,E1 29406.176,E2 29406.176} C_VEL
LIN {X 0,Y 616.238,Z 1061.094,A -85,B 0,C 180,E1 29405.193,E2 29405.193} C_VEL
LIN {X 0,Y 617.203,Z 1040.498,A -85,B 0,C 180,E1 29404.37,E2 29404.37} C_VEL
LIN {X 0,Y 618.19,Z 1017.792,A -85,B 0,C 180,E1 29403.645,E2 29403.645} C_VEL
LIN {X 0,Y 618.949,Z 995.75,A -85,B 0,C 180,E1 29403.109,E2 29403.109} C_VEL
LIN {X 0,Y 619.562,Z 972.273,A -85,B 0,C 180,E1 29402.722,E2 29402.722} C_VEL
LIN {X 0,Y 621.565,Z 842.294,A -85,B 0,C 180,E1 29401.007,E2 29401.007} C_VEL
LIN {X 0,Y 624.566,Z 724.329,A -85,B 0,C 180,E1 29399.295,E2 29399.295} C_VEL
LIN {X 0,Y 624.817,Z 708.967,A -85,B 0,C 180,E1 29399.045,E2 29399.045} C_VEL
LIN {X 0,Y 619.607,Z 680.14,A -85,B 0,C 180,E1 29398.185,E2 29398.185} C_VEL
LIN {X 0,Y 618.475,Z 674.28,A -85,B 0,C 180,E1 29397.975,E2 29397.975} C_VEL
LIN {X 0,Y 619.463,Z 658.13,A -85,B 0,C 180,E1 29396.493,E2 29396.493} C_VEL
LIN {X 0,Y 615.693,Z 643.944,A -85,B 0,C 180,E1 29394.775,E2 29394.775} C_VEL
LIN {X 0,Y 611.603,Z 631.579,A -85,B 0,C 180,E1 29393.036,E2 29393.036} C_VEL
LIN {X 0,Y 609.056,Z 624.804,A -85,B 0,C 180,E1 29391.91,E2 29391.91} C_VEL
LIN {X 0,Y 609.076,Z 624.802,A -85,B 0,C 180,E1 29388.704,E2 29388.704} C_VEL
LIN {X 0,Y 609.04,Z 624.805,A -85,B 0,C 180,E1 29385.576,E2 29385.576} C_VEL
LIN {X 0,Y 609.076,Z 624.802,A -85,B 0,C 180,E1 29382.434,E2 29382.434} C_VEL
LIN {X 0,Y 609.026,Z 624.807,A -85,B 0,C 180,E1 29379.327,E2 29379.327} C_VEL
LIN {X 0,Y 609.078,Z 624.8,A -85,B 0,C 180,E1 29376.229,E2 29376.229} C_VEL
LIN {X 0,Y 609.104,Z 625.001,A -85,B 0,C 180,E1 29374.099,E2 29374.099} C_VEL
LIN {X 0,Y 612.6,Z 634.773,A -85,B 0,C 180,E1 29372.352,E2 29372.352} C_VEL
LIN {X 0,Y 621.927,Z 650.782,A -85,B 0,C 180,E1 29371.338,E2 29371.338} C_VEL
LIN {X 0,Y 625.901,Z 659.14,A -85,B 0,C 180,E1 29370.923,E2 29370.923} C_VEL
LIN {X 0,Y 622.613,Z 770.683,A -85,B 0,C 180,E1 29369.249,E2 29369.249} C_VEL
LIN {X 0,Y 620.367,Z 888.273,A -85,B 0,C 180,E1 29367.646,E2 29367.646} C_VEL
LIN {X 0,Y 619.648,Z 933.737,A -85,B 0,C 180,E1 29367.026,E2 29367.026} C_VEL
LIN {X 0,Y 619.039,Z 956.34,A -85,B 0,C 180,E1 29366.547,E2 29366.547} C_VEL
LIN {X 0,Y 618.237,Z 977.736,A -85,B 0,C 180,E1 29365.922,E2 29365.922} C_VEL
LIN {X 0,Y 617.26,Z 999.512,A -85,B 0,C 180,E1 29365.106,E2 29365.106} C_VEL
LIN {X 0,Y 616.241,Z 1019.43,A -85,B 0,C 180,E1 29364.187,E2 29364.187} C_VEL
LIN {X 0,Y 615.12,Z 1038.622,A -85,B 0,C 180,E1 29363.116,E2 29363.116} C_VEL
LIN {X 0,Y 614.01,Z 1056.258,A -85,B 0,C 180,E1 29361.948,E2 29361.948} C_VEL
LIN {X 0,Y 612.899,Z 1073.264,A -85,B 0,C 180,E1 29360.635,E2 29360.635} C_VEL
LIN {X 0,Y 611.858,Z 1088.846,A -85,B 0,C 180,E1 29359.227,E2 29359.227} C_VEL
LIN {X 0,Y 610.904,Z 1103.187,A -85,B 0,C 180,E1 29357.714,E2 29357.714} C_VEL
LIN {X 0,Y 610.06,Z 1116.524,A -85,B 0,C 180,E1 29356.082,E2 29356.082} C_VEL
LIN {X 0,Y 609.35,Z 1128.542,A -85,B 0,C 180,E1 29354.348,E2 29354.348} C_VEL
LIN {X 0,Y 608.805,Z 1139.152,A -85,B 0,C 180,E1 29352.523,E2 29352.523} C_VEL
LIN {X 0,Y 608.38,Z 1148.818,A -85,B 0,C 180,E1 29350.513,E2 29350.513} C_VEL
LIN {X 0,Y 608.135,Z 1156.25,A -85,B 0,C 180,E1 29348.607,E2 29348.607} C_VEL
LIN {X 0,Y 607.994,Z 1162.188,A -85,B 0,C 180,E1 29346.612,E2 29346.612} C_VEL
LIN {X 0,Y 607.936,Z 1166.69,A -85,B 0,C 180,E1 29344.53,E2 29344.53} C_VEL
LIN {X 0,Y 607.914,Z 1169.448,A -85,B 0,C 180,E1 29342.547,E2 29342.547} C_VEL
LIN {X 0,Y 607.906,Z 1170.592,A -85,B 0,C 180,E1 29340.567,E2 29340.567} C_VEL
LIN {X 0,Y 607.907,Z 1170.287,A -85,B 0,C 180,E1 29338.494,E2 29338.494} C_VEL
LIN {X 0,Y 607.924,Z 1168.416,A -85,B 0,C 180,E1 29336.513,E2 29336.513} C_VEL
LIN {X 0,Y 607.958,Z 1164.812,A -85,B 0,C 180,E1 29334.434,E2 29334.434} C_VEL
LIN {X 0,Y 608.048,Z 1159.811,A -85,B 0,C 180,E1 29332.443,E2 29332.443} C_VEL
LIN {X 0,Y 608.235,Z 1152.986,A -85,B 0,C 180,E1 29330.445,E2 29330.445} C_VEL
LIN {X 0,Y 608.552,Z 1144.344,A -85,B 0,C 180,E1 29328.439,E2 29328.439} C_VEL
LIN {X 0,Y 609.023,Z 1134.232,A -85,B 0,C 180,E1 29326.521,E2 29326.521} C_VEL
LIN {X 0,Y 609.687,Z 1122.369,A -85,B 0,C 180,E1 29324.65,E2 29324.65} C_VEL
LIN {X 0,Y 610.534,Z 1108.807,A -85,B 0,C 180,E1 29322.857,E2 29322.857} C_VEL
LIN {X 0,Y 611.511,Z 1094.162,A -85,B 0,C 180,E1 29321.212,E2 29321.212} C_VEL
LIN {X 0,Y 612.642,Z 1078.048,A -85,B 0,C 180,E1 29319.66,E2 29319.66} C_VEL
LIN {X 0,Y 613.843,Z 1060.96,A -85,B 0,C 180,E1 29318.252,E2 29318.252} C_VEL
LIN {X 0,Y 615.078,Z 1042.8,A -85,B 0,C 180,E1 29316.988,E2 29316.988} C_VEL
LIN {X 0,Y 616.339,Z 1023,A -85,B 0,C 180,E1 29315.821,E2 29315.821} C_VEL
LIN {X 0,Y 617.54,Z 1003.02,A -85,B 0,C 180,E1 29314.838,E2 29314.838} C_VEL
LIN {X 0,Y 618.58,Z 982.707,A -85,B 0,C 180,E1 29314.023,E2 29314.023} C_VEL
LIN {X 0,Y 619.515,Z 961.433,A -85,B 0,C 180,E1 29313.35,E2 29313.35} C_VEL
LIN {X 0,Y 620.259,Z 939.313,A -85,B 0,C 180,E1 29312.821,E2 29312.821} C_VEL
LIN {X 0,Y 620.813,Z 916.879,A -85,B 0,C 180,E1 29312.455,E2 29312.455} C_VEL
LIN {X 0,Y 624.235,Z 703.967,A -85,B 0,C 180,E1 29309.707,E2 29309.707} C_VEL
LIN {X 0,Y 624.995,Z 663.512,A -85,B 0,C 180,E1 29309.173,E2 29309.173} C_VEL
LIN {X 0,Y 624.245,Z 660.179,A -85,B 0,C 180,E1 29309.085,E2 29309.085} C_VEL
LIN {X 0,Y 621.509,Z 656.414,A -85,B 0,C 180,E1 29308.882,E2 29308.882} C_VEL
LIN {X 0,Y 613.047,Z 649.259,A -85,B 0,C 180,E1 29308.306,E2 29308.306} C_VEL
LIN {X 0,Y 611.406,Z 646.9,A -85,B 0,C 180,E1 29308.177,E2 29308.177} C_VEL
LIN {X 0,Y 601.416,Z 627.358,A -85,B 0,C 180,E1 29307.274,E2 29307.274} C_VEL
LIN {X 0,Y 601.077,Z 625.799,A -85,B 0,C 180,E1 29307.049,E2 29307.049} C_VEL
LIN {X 0,Y 601.08,Z 625.793,A -85,B 0,C 180,E1 29303.808,E2 29303.808} C_VEL
LIN {X 0,Y 601.135,Z 625.787,A -85,B 0,C 180,E1 29300.801,E2 29300.801} C_VEL
LIN {X 0,Y 601.132,Z 625.79,A -85,B 0,C 180,E1 29297.525,E2 29297.525} C_VEL
LIN {X 0,Y 601.127,Z 625.786,A -85,B 0,C 180,E1 29294.316,E2 29294.316} C_VEL
LIN {X 0,Y 601.066,Z 625.795,A -85,B 0,C 180,E1 29291.206,E2 29291.206} C_VEL
LIN {X 0,Y 601.129,Z 625.79,A -85,B 0,C 180,E1 29288.106,E2 29288.106} C_VEL
LIN {X 0,Y 601.089,Z 625.79,A -85,B 0,C 180,E1 29285.023,E2 29285.023} C_VEL
LIN {X 0,Y 601.135,Z 625.784,A -85,B 0,C 180,E1 29281.798,E2 29281.798} C_VEL
LIN {X 0,Y 601.114,Z 625.792,A -85,B 0,C 180,E1 29278.572,E2 29278.572} C_VEL
LIN {X 0,Y 601.139,Z 625.787,A -85,B 0,C 180,E1 29275.414,E2 29275.414} C_VEL
LIN {X 0,Y 601.057,Z 625.792,A -85,B 0,C 180,E1 29272.394,E2 29272.394} C_VEL
LIN {X 0,Y 601.087,Z 625.789,A -85,B 0,C 180,E1 29269.127,E2 29269.127} C_VEL
LIN {X 0,Y 601.132,Z 625.793,A -85,B 0,C 180,E1 29266.03,E2 29266.03} C_VEL
LIN {X 0,Y 601.12,Z 625.783,A -85,B 0,C 180,E1 29262.782,E2 29262.782} C_VEL
LIN {X 0,Y 601.11,Z 625.785,A -85,B 0,C 180,E1 29259.673,E2 29259.673} C_VEL
LIN {X 0,Y 601.086,Z 625.793,A -85,B 0,C 180,E1 29256.4,E2 29256.4} C_VEL
LIN {X 0,Y 601.084,Z 625.792,A -85,B 0,C 180,E1 29253.434,E2 29253.434} C_VEL
LIN {X 0,Y 601.076,Z 625.791,A -85,B 0,C 180,E1 29250.287,E2 29250.287} C_VEL
LIN {X 0,Y 601.135,Z 625.781,A -85,B 0,C 180,E1 29247.237,E2 29247.237} C_VEL
LIN {X 0,Y 601.134,Z 625.787,A -85,B 0,C 180,E1 29243.986,E2 29243.986} C_VEL
LIN {X 0,Y 601.136,Z 625.784,A -85,B 0,C 180,E1 29240.717,E2 29240.717} C_VEL
LIN {X 0,Y 601.066,Z 625.787,A -85,B 0,C 180,E1 29237.61,E2 29237.61} C_VEL
LIN {X 0,Y 601.115,Z 625.791,A -85,B 0,C 180,E1 29234.468,E2 29234.468} C_VEL
LIN {X 0,Y 601.092,Z 625.791,A -85,B 0,C 180,E1 29231.376,E2 29231.376} C_VEL
LIN {X 0,Y 601.122,Z 625.785,A -85,B 0,C 180,E1 29228.126,E2 29228.126} C_VEL
LIN {X 0,Y 601.115,Z 625.789,A -85,B 0,C 180,E1 29225.009,E2 29225.009} C_VEL
LIN {X 0,Y 601.141,Z 625.79,A -85,B 0,C 180,E1 29221.813,E2 29221.813} C_VEL
LIN {X 0,Y 601.062,Z 625.794,A -85,B 0,C 180,E1 29218.847,E2 29218.847} C_VEL
LIN {X 0,Y 601.077,Z 625.793,A -85,B 0,C 180,E1 29215.559,E2 29215.559} C_VEL
LIN {X 0,Y 601.13,Z 625.793,A -85,B 0,C 180,E1 29212.501,E2 29212.501} C_VEL
LIN {X 0,Y 601.118,Z 625.789,A -85,B 0,C 180,E1 29209.307,E2 29209.307} C_VEL
LIN {X 0,Y 601.112,Z 625.788,A -85,B 0,C 180,E1 29206.209,E2 29206.209} C_VEL
LIN {X 0,Y 601.095,Z 625.795,A -85,B 0,C 180,E1 29202.956,E2 29202.956} C_VEL
LIN {X 0,Y 601.112,Z 625.904,A -85,B 0,C 180,E1 29201.212,E2 29201.212} C_VEL
LIN {X 0,Y 607.356,Z 649.066,A -85,B 0,C 180,E1 29199.161,E2 29199.161} C_VEL
LIN {X 0,Y 606.569,Z 693.739,A -85,B 0,C 180,E1 29195.755,E2 29195.755} C_VEL
LIN {X 0,Y 605.858,Z 734.469,A -85,B 0,C 180,E1 29192.658,E2 29192.658} C_VEL
LIN {X 0,Y 605.007,Z 775.951,A -85,B 0,C 180,E1 29189.502,E2 29189.502} C_VEL
LIN {X 0,Y 604.219,Z 817.698,A -85,B 0,C 180,E1 29186.324,E2 29186.324} C_VEL
LIN {X 0,Y 604.111,Z 826.175,A -85,B 0,C 180,E1 29185.706,E2 29185.706} C_VEL
LIN {X 0,Y 604.454,Z 833.643,A -85,B 0,C 180,E1 29185.597,E2 29185.597} C_VEL
LIN {X 0,Y 603.345,Z 968.863,A -85,B 0,C 180,E1 29183.837,E2 29183.837} C_VEL
LIN {X 0,Y 603.209,Z 985.147,A -85,B 0,C 180,E1 29183.446,E2 29183.446} C_VEL
LIN {X 0,Y 602.974,Z 1001.163,A -85,B 0,C 180,E1 29182.881,E2 29182.881} C_VEL
LIN {X 0,Y 602.657,Z 1015.85,A -85,B 0,C 180,E1 29182.173,E2 29182.173} C_VEL
LIN {X 0,Y 602.321,Z 1029.767,A -85,B 0,C 180,E1 29181.316,E2 29181.316} C_VEL
LIN {X 0,Y 601.929,Z 1042.63,A -85,B 0,C 180,E1 29180.312,E2 29180.312} C_VEL
LIN {X 0,Y 601.579,Z 1054.021,A -85,B 0,C 180,E1 29179.211,E2 29179.211} C_VEL
LIN {X 0,Y 601.242,Z 1064.288,A -85,B 0,C 180,E1 29177.97,E2 29177.97} C_VEL
LIN {X 0,Y 600.973,Z 1073.239,A -85,B 0,C 180,E1 29176.605,E2 29176.605} C_VEL
LIN {X 0,Y 600.781,Z 1080.083,A -85,B 0,C 180,E1 29175.243,E2 29175.243} C_VEL
LIN {X 0,Y 600.658,Z 1085.571,A -85,B 0,C 180,E1 29173.769,E2 29173.769} C_VEL
LIN {X 0,Y 600.579,Z 1089.557,A -85,B 0,C 180,E1 29172.107,E2 29172.107} C_VEL
LIN {X 0,Y 600.561,Z 1091.398,A -85,B 0,C 180,E1 29170.55,E2 29170.55} C_VEL
LIN {X 0,Y 600.593,Z 1091.344,A -85,B 0,C 180,E1 29169.001,E2 29169.001} C_VEL
LIN {X 0,Y 600.667,Z 1089.542,A -85,B 0,C 180,E1 29167.458,E2 29167.458} C_VEL
LIN {X 0,Y 600.784,Z 1085.823,A -85,B 0,C 180,E1 29165.921,E2 29165.921} C_VEL
LIN {X 0,Y 600.97,Z 1080.586,A -85,B 0,C 180,E1 29164.483,E2 29164.483} C_VEL
LIN {X 0,Y 601.222,Z 1073.346,A -85,B 0,C 180,E1 29163.049,E2 29163.049} C_VEL
LIN {X 0,Y 601.547,Z 1064.608,A -85,B 0,C 180,E1 29161.712,E2 29161.712} C_VEL
LIN {X 0,Y 601.93,Z 1054.205,A -85,B 0,C 180,E1 29160.471,E2 29160.471} C_VEL
LIN {X 0,Y 602.329,Z 1042.82,A -85,B 0,C 180,E1 29159.38,E2 29159.38} C_VEL
LIN {X 0,Y 602.725,Z 1029.687,A -85,B 0,C 180,E1 29158.382,E2 29158.382} C_VEL
LIN {X 0,Y 603.033,Z 1016.374,A -85,B 0,C 180,E1 29157.575,E2 29157.575} C_VEL
LIN {X 0,Y 603.312,Z 1002.06,A -85,B 0,C 180,E1 29156.91,E2 29156.91} C_VEL
LIN {X 0,Y 603.51,Z 987.924,A -85,B 0,C 180,E1 29156.418,E2 29156.418} C_VEL
LIN {X 0,Y 603.609,Z 972.827,A -85,B 0,C 180,E1 29156.038,E2 29156.038} C_VEL
LIN {X 0,Y 603.796,Z 932.558,A -85,B 0,C 180,E1 29155.488,E2 29155.488} C_VEL
LIN {X 0,Y 605.034,Z 830.241,A -85,B 0,C 180,E1 29154.093,E2 29154.093} C_VEL
LIN {X 0,Y 605.741,Z 791.051,A -85,B 0,C 180,E1 29151.168,E2 29151.168} C_VEL
LIN {X 0,Y 606.314,Z 751.641,A -85,B 0,C 180,E1 29148.248,E2 29148.248} C_VEL
LIN {X 0,Y 606.805,Z 708.921,A -85,B 0,C 180,E1 29145.152,E2 29145.152} C_VEL
LIN {X 0,Y 606.993,Z 662.475,A -85,B 0,C 180,E1 29141.858,E2 29141.858} C_VEL
LIN {X 0,Y 606.873,Z 645.179,A -85,B 0,C 180,E1 29140.658,E2 29140.658} C_VEL
LIN {X 0,Y 601.719,Z 628.046,A -85,B 0,C 180,E1 29139.224,E2 29139.224} C_VEL
LIN {X 0,Y 601.099,Z 625.796,A -85,B 0,C 180,E1 29139.02,E2 29139.02} C_VEL
LIN {X 0,Y 601.127,Z 625.798,A -85,B 0,C 180,E1 29135.944,E2 29135.944} C_VEL
LIN {X 0,Y 601.121,Z 625.793,A -85,B 0,C 180,E1 29132.777,E2 29132.777} C_VEL
LIN {X 0,Y 601.133,Z 625.789,A -85,B 0,C 180,E1 29129.402,E2 29129.402} C_VEL
LIN {X 0,Y 601.127,Z 625.791,A -85,B 0,C 180,E1 29126.134,E2 29126.134} C_VEL
LIN {X 0,Y 601.108,Z 625.794,A -85,B 0,C 180,E1 29122.974,E2 29122.974} C_VEL
LIN {X 0,Y 601.112,Z 625.791,A -85,B 0,C 180,E1 29119.918,E2 29119.918} C_VEL
LIN {X 0,Y 601.127,Z 625.788,A -85,B 0,C 180,E1 29116.608,E2 29116.608} C_VEL
LIN {X 0,Y 601.141,Z 625.789,A -85,B 0,C 180,E1 29113.374,E2 29113.374} C_VEL
LIN {X 0,Y 601.095,Z 625.794,A -85,B 0,C 180,E1 29110.194,E2 29110.194} C_VEL
LIN {X 0,Y 601.137,Z 625.884,A -85,B 0,C 180,E1 29107.805,E2 29107.805} C_VEL
LIN {X 0,Y 609.489,Z 651.708,A -85,B 0,C 180,E1 29104.811,E2 29104.811} C_VEL
LIN {X 0,Y 612.506,Z 662.42,A -85,B 0,C 180,E1 29103.636,E2 29103.636} C_VEL
LIN {X 0,Y 611.525,Z 680.435,A -85,B 0,C 180,E1 29102.075,E2 29102.075} C_VEL
LIN {X 0,Y 617.9,Z 712.176,A -85,B 0,C 180,E1 29101.248,E2 29101.248} C_VEL
LIN {X 0,Y 613.655,Z 953.925,A -85,B 0,C 180,E1 29098.059,E2 29098.059} C_VEL
LIN {X 0,Y 612.961,Z 988.32,A -85,B 0,C 180,E1 29097.574,E2 29097.574} C_VEL
LIN {X 0,Y 612.156,Z 1010.026,A -85,B 0,C 180,E1 29097.109,E2 29097.109} C_VEL
LIN {X 0,Y 611.16,Z 1031.487,A -85,B 0,C 180,E1 29096.474,E2 29096.474} C_VEL
LIN {X 0,Y 609.956,Z 1053.526,A -85,B 0,C 180,E1 29095.642,E2 29095.642} C_VEL
LIN {X 0,Y 608.721,Z 1073.882,A -85,B 0,C 180,E1 29094.693,E2 29094.693} C_VEL
LIN {X 0,Y 607.417,Z 1093.669,A -85,B 0,C 180,E1 29093.577,E2 29093.577} C_VEL
LIN {X 0,Y 606.129,Z 1112.062,A -85,B 0,C 180,E1 29092.347,E2 29092.347} C_VEL
LIN {X 0,Y 604.838,Z 1130.299,A -85,B 0,C 180,E1 29090.919,E2 29090.919} C_VEL
LIN {X 0,Y 603.734,Z 1146.507,A -85,B 0,C 180,E1 29089.443,E2 29089.443} C_VEL
LIN {X 0,Y 602.735,Z 1161.215,A -85,B 0,C 180,E1 29087.871,E2 29087.871} C_VEL
LIN {X 0,Y 601.855,Z 1175.443,A -85,B 0,C 180,E1 29086.106,E2 29086.106} C_VEL
LIN {X 0,Y 601.18,Z 1187.603,A -85,B 0,C 180,E1 29084.347,E2 29084.347} C_VEL
LIN {X 0,Y 600.668,Z 1198.298,A -85,B 0,C 180,E1 29082.496,E2 29082.496} C_VEL
LIN {X 0,Y 600.315,Z 1207.655,A -85,B 0,C 180,E1 29080.556,E2 29080.556} C_VEL
LIN {X 0,Y 600.107,Z 1215.281,A -85,B 0,C 180,E1 29078.623,E2 29078.623} C_VEL
LIN {X 0,Y 599.976,Z 1221.242,A -85,B 0,C 180,E1 29076.647,E2 29076.647} C_VEL
LIN {X 0,Y 599.934,Z 1225.963,A -85,B 0,C 180,E1 29074.491,E2 29074.491} C_VEL
LIN {X 0,Y 599.922,Z 1228.752,A -85,B 0,C 180,E1 29072.482,E2 29072.482} C_VEL
LIN {X 0,Y 599.912,Z 1229.836,A -85,B 0,C 180,E1 29070.476,E2 29070.476} C_VEL
LIN {X 0,Y 599.916,Z 1229.36,A -85,B 0,C 180,E1 29068.375,E2 29068.375} C_VEL
LIN {X 0,Y 599.926,Z 1227.319,A -85,B 0,C 180,E1 29066.368,E2 29066.368} C_VEL
LIN {X 0,Y 599.949,Z 1223.591,A -85,B 0,C 180,E1 29064.356,E2 29064.356} C_VEL
LIN {X 0,Y 600.025,Z 1218.239,A -85,B 0,C 180,E1 29062.338,E2 29062.338} C_VEL
LIN {X 0,Y 600.187,Z 1211.441,A -85,B 0,C 180,E1 29060.409,E2 29060.409} C_VEL
LIN {X 0,Y 600.484,Z 1202.38,A -85,B 0,C 180,E1 29058.375,E2 29058.375} C_VEL
LIN {X 0,Y 600.93,Z 1191.754,A -85,B 0,C 180,E1 29056.43,E2 29056.43} C_VEL
LIN {X 0,Y 601.534,Z 1179.62,A -85,B 0,C 180,E1 29054.575,E2 29054.575} C_VEL
LIN {X 0,Y 602.283,Z 1165.845,A -85,B 0,C 180,E1 29052.811,E2 29052.811} C_VEL
LIN {X 0,Y 603.203,Z 1150.552,A -85,B 0,C 180,E1 29051.14,E2 29051.14} C_VEL
LIN {X 0,Y 604.228,Z 1134.259,A -85,B 0,C 180,E1 29049.613,E2 29049.613} C_VEL
LIN {X 0,Y 605.308,Z 1117.009,A -85,B 0,C 180,E1 29048.231,E2 29048.231} C_VEL
LIN {X 0,Y 606.422,Z 1098.951,A -85,B 0,C 180,E1 29046.996,E2 29046.996} C_VEL
LIN {X 0,Y 607.647,Z 1078.517,A -85,B 0,C 180,E1 29045.811,E2 29045.811} C_VEL
LIN {X 0,Y 608.778,Z 1058.212,A -85,B 0,C 180,E1 29044.823,E2 29044.823} C_VEL
LIN {X 0,Y 609.85,Z 1036.808,A -85,B 0,C 180,E1 29043.98,E2 29043.98} C_VEL
LIN {X 0,Y 610.814,Z 1014.622,A -85,B 0,C 180,E1 29043.287,E2 29043.287} C_VEL
LIN {X 0,Y 611.689,Z 991.294,A -85,B 0,C 180,E1 29042.744,E2 29042.744} C_VEL
LIN {X 0,Y 612.284,Z 967.777,A -85,B 0,C 180,E1 29042.367,E2 29042.367} C_VEL
LIN {X 0,Y 614.346,Z 848.254,A -85,B 0,C 180,E1 29040.746,E2 29040.746} C_VEL
LIN {X 0,Y 617.531,Z 734.485,A -85,B 0,C 180,E1 29039.049,E2 29039.049} C_VEL
LIN {X 0,Y 618.122,Z 710.49,A -85,B 0,C 180,E1 29038.657,E2 29038.657} C_VEL
LIN {X 0,Y 612.892,Z 680.722,A -85,B 0,C 180,E1 29037.73,E2 29037.73} C_VEL
LIN {X 0,Y 611.448,Z 673.365,A -85,B 0,C 180,E1 29037.451,E2 29037.451} C_VEL
LIN {X 0,Y 612.229,Z 660.862,A -85,B 0,C 180,E1 29036.269,E2 29036.269} C_VEL
LIN {X 0,Y 608.832,Z 647.79,A -85,B 0,C 180,E1 29034.637,E2 29034.637} C_VEL
LIN {X 0,Y 604.883,Z 635.758,A -85,B 0,C 180,E1 29032.889,E2 29032.889} C_VEL
LIN {X 0,Y 601.953,Z 628.507,A -85,B 0,C 180,E1 29031.633,E2 29031.633} C_VEL
LIN {X 0,Y 601.122,Z 625.791,A -85,B 0,C 180,E1 29031.121,E2 29031.121} C_VEL
LIN {X 0,Y 601.117,Z 625.794,A -85,B 0,C 180,E1 29027.893,E2 29027.893} C_VEL
LIN {X 0,Y 601.134,Z 625.79,A -85,B 0,C 180,E1 29024.718,E2 29024.718} C_VEL
LIN {X 0,Y 601.097,Z 625.795,A -85,B 0,C 180,E1 29021.534,E2 29021.534} C_VEL
LIN {X 0,Y 601.141,Z 625.791,A -85,B 0,C 180,E1 29018.424,E2 29018.424} C_VEL
LIN {X 0,Y 601.082,Z 625.796,A -85,B 0,C 180,E1 29015.236,E2 29015.236} C_VEL
LIN {X 0,Y 601.096,Z 625.847,A -85,B 0,C 180,E1 29014.959,E2 29014.959} C_VEL
LIN {X 0,Y 603.836,Z 633.495,A -85,B 0,C 180,E1 29013.428,E2 29013.428} C_VEL
LIN {X 0,Y 604.885,Z 636.065,A -85,B 0,C 180,E1 29012.974,E2 29012.974} C_VEL
LIN {X 0,Y 612.459,Z 648.491,A -85,B 0,C 180,E1 29012.079,E2 29012.079} C_VEL
LIN {X 0,Y 618.713,Z 660.208,A -85,B 0,C 180,E1 29011.383,E2 29011.383} C_VEL
LIN {X 0,Y 619.289,Z 662.045,A -85,B 0,C 180,E1 29011.309,E2 29011.309} C_VEL
LIN {X 0,Y 615.583,Z 774.863,A -85,B 0,C 180,E1 29009.561,E2 29009.561} C_VEL
LIN {X 0,Y 613.146,Z 887.543,A -85,B 0,C 180,E1 29007.975,E2 29007.975} C_VEL
LIN {X 0,Y 612.324,Z 934.39,A -85,B 0,C 180,E1 29007.321,E2 29007.321} C_VEL
LIN {X 0,Y 611.672,Z 957.205,A -85,B 0,C 180,E1 29006.827,E2 29006.827} C_VEL
LIN {X 0,Y 610.838,Z 978.123,A -85,B 0,C 180,E1 29006.205,E2 29006.205} C_VEL
LIN {X 0,Y 609.809,Z 999.841,A -85,B 0,C 180,E1 29005.382,E2 29005.382} C_VEL
LIN {X 0,Y 608.737,Z 1019.754,A -85,B 0,C 180,E1 29004.453,E2 29004.453} C_VEL
LIN {X 0,Y 607.553,Z 1038.944,A -85,B 0,C 180,E1 29003.369,E2 29003.369} C_VEL
LIN {X 0,Y 606.385,Z 1056.6,A -85,B 0,C 180,E1 29002.187,E2 29002.187} C_VEL
LIN {X 0,Y 605.171,Z 1074.198,A -85,B 0,C 180,E1 29000.809,E2 29000.809} C_VEL
LIN {X 0,Y 604.052,Z 1090.273,A -85,B 0,C 180,E1 28999.335,E2 28999.335} C_VEL
LIN {X 0,Y 603.032,Z 1104.796,A -85,B 0,C 180,E1 28997.765,E2 28997.765} C_VEL
LIN {X 0,Y 602.098,Z 1118.742,A -85,B 0,C 180,E1 28996.004,E2 28996.004} C_VEL
LIN {X 0,Y 601.367,Z 1130.729,A -85,B 0,C 180,E1 28994.221,E2 28994.221} C_VEL
LIN {X 0,Y 600.801,Z 1141.445,A -85,B 0,C 180,E1 28992.302,E2 28992.302} C_VEL
LIN {X 0,Y 600.397,Z 1150.336,A -85,B 0,C 180,E1 28990.364,E2 28990.364} C_VEL
LIN {X 0,Y 600.143,Z 1157.826,A -85,B 0,C 180,E1 28988.336,E2 28988.336} C_VEL
LIN {X 0,Y 600.008,Z 1163.555,A -85,B 0,C 180,E1 28986.316,E2 28986.316} C_VEL
LIN {X 0,Y 599.942,Z 1167.56,A -85,B 0,C 180,E1 28984.303,E2 28984.303} C_VEL
LIN {X 0,Y 599.916,Z 1170.155,A -85,B 0,C 180,E1 28982.199,E2 28982.199} C_VEL
LIN {X 0,Y 599.916,Z 1171.075,A -85,B 0,C 180,E1 28980.193,E2 28980.193} C_VEL
LIN {X 0,Y 599.923,Z 1170.397,A -85,B 0,C 180,E1 28978.092,E2 28978.092} C_VEL
LIN {X 0,Y 599.928,Z 1168.131,A -85,B 0,C 180,E1 28975.988,E2 28975.988} C_VEL
LIN {X 0,Y 599.973,Z 1164.529,A -85,B 0,C 180,E1 28974.071,E2 28974.071} C_VEL
LIN {X 0,Y 600.095,Z 1158.892,A -85,B 0,C 180,E1 28971.957,E2 28971.957} C_VEL
LIN {X 0,Y 600.32,Z 1152.184,A -85,B 0,C 180,E1 28970.027,E2 28970.027} C_VEL
LIN {X 0,Y 600.667,Z 1143.636,A -85,B 0,C 180,E1 28968.09,E2 28968.09} C_VEL
LIN {X 0,Y 601.199,Z 1133.231,A -85,B 0,C 180,E1 28966.146,E2 28966.146} C_VEL
LIN {X 0,Y 601.913,Z 1121.395,A -85,B 0,C 180,E1 28964.292,E2 28964.292} C_VEL
LIN {X 0,Y 602.822,Z 1107.872,A -85,B 0,C 180,E1 28962.506,E2 28962.506} C_VEL
LIN {X 0,Y 603.85,Z 1093.187,A -85,B 0,C 180,E1 28960.864,E2 28960.864} C_VEL
LIN {X 0,Y 605.081,Z 1076.639,A -85,B 0,C 180,E1 28959.279,E2 28959.279} C_VEL
LIN {X 0,Y 606.31,Z 1060.076,A -85,B 0,C 180,E1 28957.916,E2 28957.916} C_VEL
LIN {X 0,Y 607.625,Z 1041.745,A -85,B 0,C 180,E1 28956.638,E2 28956.638} C_VEL
LIN {X 0,Y 608.909,Z 1022.548,A -85,B 0,C 180,E1 28955.507,E2 28955.507} C_VEL
LIN {X 0,Y 610.156,Z 1002.65,A -85,B 0,C 180,E1 28954.525,E2 28954.525} C_VEL
LIN {X 0,Y 611.286,Z 981.877,A -85,B 0,C 180,E1 28953.686,E2 28953.686} C_VEL
LIN {X 0,Y 612.248,Z 960.73,A -85,B 0,C 180,E1 28953.019,E2 28953.019} C_VEL
LIN {X 0,Y 613.04,Z 937.501,A -85,B 0,C 180,E1 28952.471,E2 28952.471} C_VEL
LIN {X 0,Y 613.623,Z 913.813,A -85,B 0,C 180,E1 28952.097,E2 28952.097} C_VEL
LIN {X 0,Y 617.356,Z 699.508,A -85,B 0,C 180,E1 28949.283,E2 28949.283} C_VEL
LIN {X 0,Y 617.951,Z 660.086,A -85,B 0,C 180,E1 28948.744,E2 28948.744} C_VEL
LIN {X 0,Y 611.406,Z 646.9,A -85,B 0,C 180,E1 28948.177,E2 28948.177} C_VEL
LIN {X 0,Y 608.47,Z 643.284,A -85,B 0,C 180,E1 28947.952,E2 28947.952} C_VEL
LIN {X 0,Y 598.345,Z 636.079,A -85,B 0,C 180,E1 28947.249,E2 28947.249} C_VEL
LIN {X 0,Y 595.909,Z 632.894,A -85,B 0,C 180,E1 28947.055,E2 28947.055} C_VEL
LIN {X 0,Y 593.322,Z 627.648,A -85,B 0,C 180,E1 28946.794,E2 28946.794} C_VEL
LIN {X 0,Y 593.177,Z 626.783,A -85,B 0,C 180,E1 28946.669,E2 28946.669} C_VEL
LIN {X 0,Y 593.146,Z 626.781,A -85,B 0,C 180,E1 28943.486,E2 28943.486} C_VEL
LIN {X 0,Y 593.188,Z 626.773,A -85,B 0,C 180,E1 28940.233,E2 28940.233} C_VEL
LIN {X 0,Y 593.179,Z 626.778,A -85,B 0,C 180,E1 28937.019,E2 28937.019} C_VEL
LIN {X 0,Y 593.199,Z 626.778,A -85,B 0,C 180,E1 28933.831,E2 28933.831} C_VEL
LIN {X 0,Y 593.127,Z 626.783,A -85,B 0,C 180,E1 28930.811,E2 28930.811} C_VEL
LIN {X 0,Y 593.133,Z 626.781,A -85,B 0,C 180,E1 28927.444,E2 28927.444} C_VEL
LIN {X 0,Y 593.196,Z 626.78,A -85,B 0,C 180,E1 28924.381,E2 28924.381} C_VEL
LIN {X 0,Y 593.183,Z 626.779,A -85,B 0,C 180,E1 28921.102,E2 28921.102} C_VEL
LIN {X 0,Y 593.197,Z 626.775,A -85,B 0,C 180,E1 28917.835,E2 28917.835} C_VEL
LIN {X 0,Y 593.141,Z 626.783,A -85,B 0,C 180,E1 28914.607,E2 28914.607} C_VEL
LIN {X 0,Y 593.173,Z 626.782,A -85,B 0,C 180,E1 28911.457,E2 28911.457} C_VEL
LIN {X 0,Y 593.142,Z 626.78,A -85,B 0,C 180,E1 28908.374,E2 28908.374} C_VEL
LIN {X 0,Y 593.172,Z 626.775,A -85,B 0,C 180,E1 28905.047,E2 28905.047} C_VEL
LIN {X 0,Y 593.183,Z 626.777,A -85,B 0,C 180,E1 28901.869,E2 28901.869} C_VEL
LIN {X 0,Y 593.191,Z 626.774,A -85,B 0,C 180,E1 28898.629,E2 28898.629} C_VEL
LIN {X 0,Y 593.144,Z 626.781,A -85,B 0,C 180,E1 28895.612,E2 28895.612} C_VEL
LIN {X 0,Y 593.117,Z 626.775,A -85,B 0,C 180,E1 28892.32,E2 28892.32} C_VEL
LIN {X 0,Y 593.202,Z 626.779,A -85,B 0,C 180,E1 28889.325,E2 28889.325} C_VEL
LIN {X 0,Y 593.177,Z 626.772,A -85,B 0,C 180,E1 28886.038,E2 28886.038} C_VEL
LIN {X 0,Y 593.202,Z 626.772,A -85,B 0,C 180,E1 28882.739,E2 28882.739} C_VEL
LIN {X 0,Y 593.148,Z 626.77,A -85,B 0,C 180,E1 28879.61,E2 28879.61} C_VEL
LIN {X 0,Y 593.181,Z 626.779,A -85,B 0,C 180,E1 28876.451,E2 28876.451} C_VEL
LIN {X 0,Y 593.132,Z 626.781,A -85,B 0,C 180,E1 28873.348,E2 28873.348} C_VEL
LIN {X 0,Y 593.169,Z 626.775,A -85,B 0,C 180,E1 28870.094,E2 28870.094} C_VEL
LIN {X 0,Y 593.19,Z 626.776,A -85,B 0,C 180,E1 28866.968,E2 28866.968} C_VEL
LIN {X 0,Y 593.197,Z 626.779,A -85,B 0,C 180,E1 28863.687,E2 28863.687} C_VEL
LIN {X 0,Y 593.151,Z 626.779,A -85,B 0,C 180,E1 28860.626,E2 28860.626} C_VEL
LIN {X 0,Y 593.119,Z 626.784,A -85,B 0,C 180,E1 28857.355,E2 28857.355} C_VEL
LIN {X 0,Y 593.189,Z 626.781,A -85,B 0,C 180,E1 28854.325,E2 28854.325} C_VEL
LIN {X 0,Y 593.165,Z 626.78,A -85,B 0,C 180,E1 28851.145,E2 28851.145} C_VEL
LIN {X 0,Y 593.193,Z 626.774,A -85,B 0,C 180,E1 28847.998,E2 28847.998} C_VEL
LIN {X 0,Y 593.168,Z 626.78,A -85,B 0,C 180,E1 28844.794,E2 28844.794} C_VEL
LIN {X 0,Y 593.201,Z 626.778,A -85,B 0,C 180,E1 28841.551,E2 28841.551} C_VEL
LIN {X 0,Y 593.208,Z 626.87,A -85,B 0,C 180,E1 28841.481,E2 28841.481} C_VEL
LIN {X 0,Y 599.79,Z 651.368,A -85,B 0,C 180,E1 28839.304,E2 28839.304} C_VEL
LIN {X 0,Y 598.913,Z 697.441,A -85,B 0,C 180,E1 28835.773,E2 28835.773} C_VEL
LIN {X 0,Y 598.119,Z 738.526,A -85,B 0,C 180,E1 28832.621,E2 28832.621} C_VEL
LIN {X 0,Y 597.261,Z 778.936,A -85,B 0,C 180,E1 28829.537,E2 28829.537} C_VEL
LIN {X 0,Y 596.456,Z 820.353,A -85,B 0,C 180,E1 28826.372,E2 28826.372} C_VEL
LIN {X 0,Y 596.38,Z 826.963,A -85,B 0,C 180,E1 28825.893,E2 28825.893} C_VEL
LIN {X 0,Y 596.712,Z 834.487,A -85,B 0,C 180,E1 28825.782,E2 28825.782} C_VEL
LIN {X 0,Y 595.533,Z 969.812,A -85,B 0,C 180,E1 28823.988,E2 28823.988} C_VEL
LIN {X 0,Y 595.392,Z 986.131,A -85,B 0,C 180,E1 28823.589,E2 28823.589} C_VEL
LIN {X 0,Y 595.142,Z 1002.303,A -85,B 0,C 180,E1 28823.008,E2 28823.008} C_VEL
LIN {X 0,Y 594.807,Z 1017.251,A -85,B 0,C 180,E1 28822.273,E2 28822.273} C_VEL
LIN {X 0,Y 594.454,Z 1031.078,A -85,B 0,C 180,E1 28821.405,E2 28821.405} C_VEL
LIN {X 0,Y 594.035,Z 1044.157,A -85,B 0,C 180,E1 28820.362,E2 28820.362} C_VEL
LIN {X 0,Y 593.679,Z 1055.213,A -85,B 0,C 180,E1 28819.273,E2 28819.273} C_VEL
LIN {X 0,Y 593.338,Z 1065.093,A -85,B 0,C 180,E1 28818.061,E2 28818.061} C_VEL
LIN {X 0,Y 593.049,Z 1074.224,A -85,B 0,C 180,E1 28816.653,E2 28816.653} C_VEL
LIN {X 0,Y 592.844,Z 1081.158,A -85,B 0,C 180,E1 28815.252,E2 28815.252} C_VEL
LIN {X 0,Y 592.717,Z 1086.625,A -85,B 0,C 180,E1 28813.758,E2 28813.758} C_VEL
LIN {X 0,Y 592.633,Z 1090.571,A -85,B 0,C 180,E1 28812.074,E2 28812.074} C_VEL
LIN {X 0,Y 592.617,Z 1092.362,A -85,B 0,C 180,E1 28810.497,E2 28810.497} C_VEL
LIN {X 0,Y 592.655,Z 1092.272,A -85,B 0,C 180,E1 28808.927,E2 28808.927} C_VEL
LIN {X 0,Y 592.737,Z 1090.415,A -85,B 0,C 180,E1 28807.364,E2 28807.364} C_VEL
LIN {X 0,Y 592.873,Z 1086.646,A -85,B 0,C 180,E1 28805.806,E2 28805.806} C_VEL
LIN {X 0,Y 593.081,Z 1081.35,A -85,B 0,C 180,E1 28804.349,E2 28804.349} C_VEL
LIN {X 0,Y 593.36,Z 1074.038,A -85,B 0,C 180,E1 28802.896,E2 28802.896} C_VEL
LIN {X 0,Y 593.685,Z 1065.901,A -85,B 0,C 180,E1 28801.639,E2 28801.639} C_VEL
LIN {X 0,Y 594.092,Z 1055.585,A -85,B 0,C 180,E1 28800.384,E2 28800.384} C_VEL
LIN {X 0,Y 594.535,Z 1043.686,A -85,B 0,C 180,E1 28799.227,E2 28799.227} C_VEL
LIN {X 0,Y 594.954,Z 1030.495,A -85,B 0,C 180,E1 28798.216,E2 28798.216} C_VEL
LIN {X 0,Y 595.282,Z 1017.11,A -85,B 0,C 180,E1 28797.399,E2 28797.399} C_VEL
LIN {X 0,Y 595.572,Z 1002.653,A -85,B 0,C 180,E1 28796.726,E2 28796.726} C_VEL
LIN {X 0,Y 595.774,Z 988.795,A -85,B 0,C 180,E1 28796.239,E2 28796.239} C_VEL
LIN {X 0,Y 595.879,Z 973.855,A -85,B 0,C 180,E1 28795.857,E2 28795.857} C_VEL
LIN {X 0,Y 596.09,Z 932.886,A -85,B 0,C 180,E1 28795.285,E2 28795.285} C_VEL
LIN {X 0,Y 597.408,Z 831.354,A -85,B 0,C 180,E1 28793.873,E2 28793.873} C_VEL
LIN {X 0,Y 598.215,Z 791.957,A -85,B 0,C 180,E1 28790.91,E2 28790.91} C_VEL
LIN {X 0,Y 598.747,Z 756.031,A -85,B 0,C 180,E1 28788.243,E2 28788.243} C_VEL
LIN {X 0,Y 599.288,Z 717.898,A -85,B 0,C 180,E1 28785.455,E2 28785.455} C_VEL
LIN {X 0,Y 599.512,Z 677.134,A -85,B 0,C 180,E1 28782.528,E2 28782.528} C_VEL
LIN {X 0,Y 599.729,Z 648.474,A -85,B 0,C 180,E1 28780.52,E2 28780.52} C_VEL
LIN {X 0,Y 594.572,Z 631.279,A -85,B 0,C 180,E1 28779.055,E2 28779.055} C_VEL
LIN {X 0,Y 593.187,Z 626.783,A -85,B 0,C 180,E1 28778.646,E2 28778.646} C_VEL
LIN {X 0,Y 593.175,Z 626.787,A -85,B 0,C 180,E1 28775.5,E2 28775.5} C_VEL
LIN {X 0,Y 593.166,Z 626.783,A -85,B 0,C 180,E1 28772.453,E2 28772.453} C_VEL
LIN {X 0,Y 593.196,Z 626.779,A -85,B 0,C 180,E1 28769.061,E2 28769.061} C_VEL
LIN {X 0,Y 593.201,Z 626.778,A -85,B 0,C 180,E1 28765.736,E2 28765.736} C_VEL
LIN {X 0,Y 593.161,Z 626.783,A -85,B 0,C 180,E1 28762.393,E2 28762.393} C_VEL
LIN {X 0,Y 593.202,Z 626.779,A -85,B 0,C 180,E1 28759.182,E2 28759.182} C_VEL
LIN {X 0,Y 593.18,Z 626.781,A -85,B 0,C 180,E1 28756.012,E2 28756.012} C_VEL
LIN {X 0,Y 593.187,Z 626.776,A -85,B 0,C 180,E1 28752.524,E2 28752.524} C_VEL
LIN {X 0,Y 593.206,Z 626.774,A -85,B 0,C 180,E1 28749.313,E2 28749.313} C_VEL
LIN {X 0,Y 593.208,Z 626.905,A -85,B 0,C 180,E1 28748.234,E2 28748.234} C_VEL
LIN {X 0,Y 601.838,Z 653.579,A -85,B 0,C 180,E1 28745.086,E2 28745.086} C_VEL
LIN {X 0,Y 605.159,Z 664.89,A -85,B 0,C 180,E1 28743.834,E2 28743.834} C_VEL
LIN {X 0,Y 604.263,Z 680.057,A -85,B 0,C 180,E1 28742.501,E2 28742.501} C_VEL
LIN {X 0,Y 610.981,Z 713.592,A -85,B 0,C 180,E1 28741.61,E2 28741.61} C_VEL
LIN {X 0,Y 606.505,Z 948.251,A -85,B 0,C 180,E1 28738.455,E2 28738.455} C_VEL
LIN {X 0,Y 605.704,Z 987.206,A -85,B 0,C 180,E1 28737.906,E2 28737.906} C_VEL
LIN {X 0,Y 604.867,Z 1008.779,A -85,B 0,C 180,E1 28737.442,E2 28737.442} C_VEL
LIN {X 0,Y 603.799,Z 1030.576,A -85,B 0,C 180,E1 28736.798,E2 28736.798} C_VEL
LIN {X 0,Y 602.571,Z 1052.231,A -85,B 0,C 180,E1 28735.979,E2 28735.979} C_VEL
LIN {X 0,Y 601.282,Z 1072.508,A -85,B 0,C 180,E1 28735.036,E2 28735.036} C_VEL
LIN {X 0,Y 599.92,Z 1092.159,A -85,B 0,C 180,E1 28733.923,E2 28733.923} C_VEL
LIN {X 0,Y 598.514,Z 1111.094,A -85,B 0,C 180,E1 28732.654,E2 28732.654} C_VEL
LIN {X 0,Y 597.199,Z 1128.948,A -85,B 0,C 180,E1 28731.251,E2 28731.251} C_VEL
LIN {X 0,Y 595.968,Z 1145.772,A -85,B 0,C 180,E1 28729.706,E2 28729.706} C_VEL
LIN {X 0,Y 594.905,Z 1160.552,A -85,B 0,C 180,E1 28728.114,E2 28728.114} C_VEL
LIN {X 0,Y 593.968,Z 1174.843,A -85,B 0,C 180,E1 28726.326,E2 28726.326} C_VEL
LIN {X 0,Y 593.259,Z 1187.056,A -85,B 0,C 180,E1 28724.543,E2 28724.543} C_VEL
LIN {X 0,Y 592.716,Z 1197.785,A -85,B 0,C 180,E1 28722.667,E2 28722.667} C_VEL
LIN {X 0,Y 592.341,Z 1207.183,A -85,B 0,C 180,E1 28720.699,E2 28720.699} C_VEL
LIN {X 0,Y 592.112,Z 1214.842,A -85,B 0,C 180,E1 28718.74,E2 28718.74} C_VEL
LIN {X 0,Y 591.979,Z 1220.948,A -85,B 0,C 180,E1 28716.691,E2 28716.691} C_VEL
LIN {X 0,Y 591.938,Z 1225.565,A -85,B 0,C 180,E1 28714.552,E2 28714.552} C_VEL
LIN {X 0,Y 591.929,Z 1228.364,A -85,B 0,C 180,E1 28712.516,E2 28712.516} C_VEL
LIN {X 0,Y 591.922,Z 1229.448,A -85,B 0,C 180,E1 28710.483,E2 28710.483} C_VEL
LIN {X 0,Y 591.926,Z 1228.96,A -85,B 0,C 180,E1 28708.353,E2 28708.353} C_VEL
LIN {X 0,Y 591.935,Z 1226.895,A -85,B 0,C 180,E1 28706.318,E2 28706.318} C_VEL
LIN {X 0,Y 591.955,Z 1223.005,A -85,B 0,C 180,E1 28704.219,E2 28704.219} C_VEL
LIN {X 0,Y 592.04,Z 1217.424,A -85,B 0,C 180,E1 28702.136,E2 28702.136} C_VEL
LIN {X 0,Y 592.212,Z 1210.508,A -85,B 0,C 180,E1 28700.18,E2 28700.18} C_VEL
LIN {X 0,Y 592.518,Z 1201.739,A -85,B 0,C 180,E1 28698.217,E2 28698.217} C_VEL
LIN {X 0,Y 592.986,Z 1190.948,A -85,B 0,C 180,E1 28696.231,E2 28696.231} C_VEL
LIN {X 0,Y 593.622,Z 1178.803,A -85,B 0,C 180,E1 28694.364,E2 28694.364} C_VEL
LIN {X 0,Y 594.361,Z 1165.739,A -85,B 0,C 180,E1 28692.675,E2 28692.675} C_VEL
LIN {X 0,Y 595.318,Z 1150.473,A -85,B 0,C 180,E1 28690.982,E2 28690.982} C_VEL
LIN {X 0,Y 596.395,Z 1134.216,A -85,B 0,C 180,E1 28689.436,E2 28689.436} C_VEL
LIN {X 0,Y 597.528,Z 1116.999,A -85,B 0,C 180,E1 28688.036,E2 28688.036} C_VEL
LIN {X 0,Y 598.746,Z 1098.173,A -85,B 0,C 180,E1 28686.731,E2 28686.731} C_VEL
LIN {X 0,Y 600.039,Z 1077.781,A -85,B 0,C 180,E1 28685.537,E2 28685.537} C_VEL
LIN {X 0,Y 601.232,Z 1057.577,A -85,B 0,C 180,E1 28684.543,E2 28684.543} C_VEL
LIN {X 0,Y 602.39,Z 1035.965,A -85,B 0,C 180,E1 28683.682,E2 28683.682} C_VEL
LIN {X 0,Y 603.404,Z 1013.792,A -85,B 0,C 180,E1 28682.981,E2 28682.981} C_VEL
LIN {X 0,Y 604.368,Z 989.983,A -85,B 0,C 180,E1 28682.423,E2 28682.423} C_VEL
LIN {X 0,Y 605.006,Z 965.907,A -85,B 0,C 180,E1 28682.034,E2 28682.034} C_VEL
LIN {X 0,Y 607.218,Z 851.846,A -85,B 0,C 180,E1 28680.441,E2 28680.441} C_VEL
LIN {X 0,Y 610.687,Z 739.869,A -85,B 0,C 180,E1 28678.718,E2 28678.718} C_VEL
LIN {X 0,Y 611.542,Z 712.025,A -85,B 0,C 180,E1 28678.248,E2 28678.248} C_VEL
LIN {X 0,Y 606.877,Z 684.053,A -85,B 0,C 180,E1 28677.346,E2 28677.346} C_VEL
LIN {X 0,Y 604.534,Z 672.403,A -85,B 0,C 180,E1 28676.89,E2 28676.89} C_VEL
LIN {X 0,Y 605.089,Z 663.825,A -85,B 0,C 180,E1 28676.053,E2 28676.053} C_VEL
LIN {X 0,Y 601.721,Z 650.653,A -85,B 0,C 180,E1 28674.351,E2 28674.351} C_VEL
LIN {X 0,Y 598.189,Z 639.886,A -85,B 0,C 180,E1 28672.718,E2 28672.718} C_VEL
LIN {X 0,Y 594.566,Z 630.359,A -85,B 0,C 180,E1 28670.984,E2 28670.984} C_VEL
LIN {X 0,Y 593.199,Z 626.779,A -85,B 0,C 180,E1 28670.233,E2 28670.233} C_VEL
LIN {X 0,Y 593.179,Z 626.781,A -85,B 0,C 180,E1 28667.02,E2 28667.02} C_VEL
LIN {X 0,Y 593.165,Z 626.784,A -85,B 0,C 180,E1 28663.683,E2 28663.683} C_VEL
LIN {X 0,Y 593.204,Z 626.779,A -85,B 0,C 180,E1 28660.518,E2 28660.518} C_VEL
LIN {X 0,Y 593.147,Z 626.783,A -85,B 0,C 180,E1 28657.365,E2 28657.365} C_VEL
LIN {X 0,Y 593.189,Z 626.82,A -85,B 0,C 180,E1 28655.917,E2 28655.917} C_VEL
LIN {X 0,Y 596.346,Z 635.492,A -85,B 0,C 180,E1 28654.001,E2 28654.001} C_VEL
LIN {X 0,Y 597.221,Z 637.493,A -85,B 0,C 180,E1 28653.641,E2 28653.641} C_VEL
LIN {X 0,Y 604.227,Z 648.453,A -85,B 0,C 180,E1 28652.746,E2 28652.746} C_VEL
LIN {X 0,Y 611.462,Z 661.429,A -85,B 0,C 180,E1 28651.89,E2 28651.89} C_VEL
LIN {X 0,Y 612.83,Z 664.704,A -85,B 0,C 180,E1 28651.721,E2 28651.721} C_VEL
LIN {X 0,Y 608.845,Z 771.281,A -85,B 0,C 180,E1 28650.006,E2 28650.006} C_VEL
LIN {X 0,Y 606.131,Z 879.027,A -85,B 0,C 180,E1 28648.427,E2 28648.427} C_VEL
LIN {X 0,Y 605.054,Z 934.83,A -85,B 0,C 180,E1 28647.632,E2 28647.632} C_VEL
LIN {X 0,Y 604.348,Z 957.868,A -85,B 0,C 180,E1 28647.124,E2 28647.124} C_VEL
LIN {X 0,Y 603.438,Z 979.367,A -85,B 0,C 180,E1 28646.472,E2 28646.472} C_VEL
LIN {X 0,Y 602.343,Z 1001.115,A -85,B 0,C 180,E1 28645.629,E2 28645.629} C_VEL
LIN {X 0,Y 601.195,Z 1021.095,A -85,B 0,C 180,E1 28644.676,E2 28644.676} C_VEL
LIN {X 0,Y 599.918,Z 1040.927,A -85,B 0,C 180,E1 28643.534,E2 28643.534} C_VEL
LIN {X 0,Y 598.63,Z 1059.11,A -85,B 0,C 180,E1 28642.279,E2 28642.279} C_VEL
LIN {X 0,Y 597.333,Z 1076.875,A -85,B 0,C 180,E1 28640.839,E2 28640.839} C_VEL
LIN {X 0,Y 596.203,Z 1092.153,A -85,B 0,C 180,E1 28639.396,E2 28639.396} C_VEL
LIN {X 0,Y 595.154,Z 1106.525,A -85,B 0,C 180,E1 28637.806,E2 28637.806} C_VEL
LIN {X 0,Y 594.217,Z 1119.788,A -85,B 0,C 180,E1 28636.09,E2 28636.09} C_VEL
LIN {X 0,Y 593.473,Z 1131.347,A -85,B 0,C 180,E1 28634.341,E2 28634.341} C_VEL
LIN {X 0,Y 592.887,Z 1141.771,A -85,B 0,C 180,E1 28632.452,E2 28632.452} C_VEL
LIN {X 0,Y 592.454,Z 1150.64,A -85,B 0,C 180,E1 28630.504,E2 28630.504} C_VEL
LIN {X 0,Y 592.185,Z 1157.882,A -85,B 0,C 180,E1 28628.547,E2 28628.547} C_VEL
LIN {X 0,Y 592.035,Z 1163.419,A -85,B 0,C 180,E1 28626.597,E2 28626.597} C_VEL
LIN {X 0,Y 591.963,Z 1167.79,A -85,B 0,C 180,E1 28624.458,E2 28624.458} C_VEL
LIN {X 0,Y 591.932,Z 1170.42,A -85,B 0,C 180,E1 28622.422,E2 28622.422} C_VEL
LIN {X 0,Y 591.924,Z 1171.425,A -85,B 0,C 180,E1 28620.389,E2 28620.389} C_VEL
LIN {X 0,Y 591.932,Z 1170.915,A -85,B 0,C 180,E1 28618.26,E2 28618.26} C_VEL
LIN {X 0,Y 591.943,Z 1168.921,A -85,B 0,C 180,E1 28616.225,E2 28616.225} C_VEL
LIN {X 0,Y 591.986,Z 1165.272,A -85,B 0,C 180,E1 28614.184,E2 28614.184} C_VEL
LIN {X 0,Y 592.11,Z 1159.79,A -85,B 0,C 180,E1 28612.043,E2 28612.043} C_VEL
LIN {X 0,Y 592.355,Z 1152.819,A -85,B 0,C 180,E1 28609.99,E2 28609.99} C_VEL
LIN {X 0,Y 592.721,Z 1144.31,A -85,B 0,C 180,E1 28608.027,E2 28608.027} C_VEL
LIN {X 0,Y 593.282,Z 1133.956,A -85,B 0,C 180,E1 28606.057,E2 28606.057} C_VEL
LIN {X 0,Y 593.993,Z 1122.881,A -85,B 0,C 180,E1 28604.278,E2 28604.278} C_VEL
LIN {X 0,Y 594.911,Z 1109.664,A -85,B 0,C 180,E1 28602.494,E2 28602.494} C_VEL
LIN {X 0,Y 596.001,Z 1095.011,A -85,B 0,C 180,E1 28600.805,E2 28600.805} C_VEL
LIN {X 0,Y 597.269,Z 1078.895,A -85,B 0,C 180,E1 28599.215,E2 28599.215} C_VEL
LIN {X 0,Y 598.601,Z 1061.795,A -85,B 0,C 180,E1 28597.772,E2 28597.772} C_VEL
LIN {X 0,Y 599.969,Z 1043.661,A -85,B 0,C 180,E1 28596.478,E2 28596.478} C_VEL
LIN {X 0,Y 601.37,Z 1023.895,A -85,B 0,C 180,E1 28595.284,E2 28595.284} C_VEL
LIN {X 0,Y 602.702,Z 1003.768,A -85,B 0,C 180,E1 28594.27,E2 28594.27} C_VEL
LIN {X 0,Y 603.885,Z 982.929,A -85,B 0,C 180,E1 28593.416,E2 28593.416} C_VEL
LIN {X 0,Y 604.904,Z 961.783,A -85,B 0,C 180,E1 28592.735,E2 28592.735} C_VEL
LIN {X 0,Y 605.731,Z 939.287,A -85,B 0,C 180,E1 28592.186,E2 28592.186} C_VEL
LIN {X 0,Y 606.343,Z 916.802,A -85,B 0,C 180,E1 28591.813,E2 28591.813} C_VEL
LIN {X 0,Y 610.19,Z 710.416,A -85,B 0,C 180,E1 28589.055,E2 28589.055} C_VEL
LIN {X 0,Y 611.085,Z 662.653,A -85,B 0,C 180,E1 28588.395,E2 28588.395} C_VEL
LIN {X 0,Y 597.481,Z 635.888,A -85,B 0,C 180,E1 28587.196,E2 28587.196} C_VEL
LIN {X 0,Y 595.909,Z 632.894,A -85,B 0,C 180,E1 28587.055,E2 28587.055} C_VEL
LIN {X 0,Y 594.005,Z 630.126,A -85,B 0,C 180,E1 28586.824,E2 28586.824} C_VEL
LIN {X 0,Y 591.58,Z 628.183,A -85,B 0,C 180,E1 28586.41,E2 28586.41} C_VEL
LIN {X 0,Y 588.663,Z 627.344,A -85,B 0,C 180,E1 28585.722,E2 28585.722} C_VEL
LIN {X 0,Y 585.763,Z 627.721,A -85,B 0,C 180,E1 28584.568,E2 28584.568} C_VEL
LIN {X 0,Y 585.203,Z 627.771,A -85,B 0,C 180,E1 28583.856,E2 28583.856} C_VEL
LIN {X 0,Y 585.26,Z 627.763,A -85,B 0,C 180,E1 28580.709,E2 28580.709} C_VEL
LIN {X 0,Y 585.255,Z 627.769,A -85,B 0,C 180,E1 28577.422,E2 28577.422} C_VEL
LIN {X 0,Y 585.258,Z 627.764,A -85,B 0,C 180,E1 28574.152,E2 28574.152} C_VEL
LIN {X 0,Y 585.185,Z 627.773,A -85,B 0,C 180,E1 28571.006,E2 28571.006} C_VEL
LIN {X 0,Y 585.226,Z 627.769,A -85,B 0,C 180,E1 28567.835,E2 28567.835} C_VEL
LIN {X 0,Y 585.235,Z 627.767,A -85,B 0,C 180,E1 28564.677,E2 28564.677} C_VEL
LIN {X 0,Y 585.239,Z 627.765,A -85,B 0,C 180,E1 28561.407,E2 28561.407} C_VEL
LIN {X 0,Y 585.235,Z 627.767,A -85,B 0,C 180,E1 28558.247,E2 28558.247} C_VEL
LIN {X 0,Y 585.223,Z 627.773,A -85,B 0,C 180,E1 28554.963,E2 28554.963} C_VEL
LIN {X 0,Y 585.208,Z 627.769,A -85,B 0,C 180,E1 28551.918,E2 28551.918} C_VEL
LIN {X 0,Y 585.193,Z 627.768,A -85,B 0,C 180,E1 28548.738,E2 28548.738} C_VEL
LIN {X 0,Y 585.263,Z 627.763,A -85,B 0,C 180,E1 28545.56,E2 28545.56} C_VEL
LIN {X 0,Y 585.254,Z 627.768,A -85,B 0,C 180,E1 28542.232,E2 28542.232} C_VEL
LIN {X 0,Y 585.261,Z 627.763,A -85,B 0,C 180,E1 28538.945,E2 28538.945} C_VEL
LIN {X 0,Y 585.194,Z 627.77,A -85,B 0,C 180,E1 28535.885,E2 28535.885} C_VEL
LIN {X 0,Y 585.196,Z 627.764,A -85,B 0,C 180,E1 28532.645,E2 28532.645} C_VEL
LIN {X 0,Y 585.231,Z 627.77,A -85,B 0,C 180,E1 28529.61,E2 28529.61} C_VEL
LIN {X 0,Y 585.232,Z 627.758,A -85,B 0,C 180,E1 28526.377,E2 28526.377} C_VEL
LIN {X 0,Y 585.24,Z 627.764,A -85,B 0,C 180,E1 28523.231,E2 28523.231} C_VEL
LIN {X 0,Y 585.23,Z 627.76,A -85,B 0,C 180,E1 28519.965,E2 28519.965} C_VEL
LIN {X 0,Y 585.221,Z 627.763,A -85,B 0,C 180,E1 28516.862,E2 28516.862} C_VEL
LIN {X 0,Y 585.183,Z 627.77,A -85,B 0,C 180,E1 28513.728,E2 28513.728} C_VEL
LIN {X 0,Y 585.26,Z 627.763,A -85,B 0,C 180,E1 28510.563,E2 28510.563} C_VEL
LIN {X 0,Y 585.259,Z 627.769,A -85,B 0,C 180,E1 28507.289,E2 28507.289} C_VEL
LIN {X 0,Y 585.259,Z 627.764,A -85,B 0,C 180,E1 28503.957,E2 28503.957} C_VEL
LIN {X 0,Y 585.202,Z 627.769,A -85,B 0,C 180,E1 28500.861,E2 28500.861} C_VEL
LIN {X 0,Y 585.203,Z 627.773,A -85,B 0,C 180,E1 28497.672,E2 28497.672} C_VEL
LIN {X 0,Y 585.226,Z 627.772,A -85,B 0,C 180,E1 28494.58,E2 28494.58} C_VEL
LIN {X 0,Y 585.226,Z 627.767,A -85,B 0,C 180,E1 28491.33,E2 28491.33} C_VEL
LIN {X 0,Y 585.247,Z 627.765,A -85,B 0,C 180,E1 28488.22,E2 28488.22} C_VEL
LIN {X 0,Y 585.234,Z 627.768,A -85,B 0,C 180,E1 28484.876,E2 28484.876} C_VEL
LIN {X 0,Y 585.251,Z 627.841,A -85,B 0,C 180,E1 28481.761,E2 28481.761} C_VEL
LIN {X 0,Y 592.186,Z 653.484,A -85,B 0,C 180,E1 28479.455,E2 28479.455} C_VEL
LIN {X 0,Y 591.307,Z 698.619,A -85,B 0,C 180,E1 28475.985,E2 28475.985} C_VEL
LIN {X 0,Y 590.451,Z 740.504,A -85,B 0,C 180,E1 28472.755,E2 28472.755} C_VEL
LIN {X 0,Y 589.519,Z 781.196,A -85,B 0,C 180,E1 28469.622,E2 28469.622} C_VEL
LIN {X 0,Y 588.695,Z 823.04,A -85,B 0,C 180,E1 28466.421,E2 28466.421} C_VEL
LIN {X 0,Y 588.654,Z 827.8,A -85,B 0,C 180,E1 28466.081,E2 28466.081} C_VEL
LIN {X 0,Y 588.966,Z 835.589,A -85,B 0,C 180,E1 28465.965,E2 28465.965} C_VEL
LIN {X 0,Y 587.711,Z 970.626,A -85,B 0,C 180,E1 28464.138,E2 28464.138} C_VEL
LIN {X 0,Y 587.565,Z 986.95,A -85,B 0,C 180,E1 28463.733,E2 28463.733} C_VEL
LIN {X 0,Y 587.308,Z 1002.88,A -85,B 0,C 180,E1 28463.156,E2 28463.156} C_VEL
LIN {X 0,Y 586.969,Z 1017.598,A -85,B 0,C 180,E1 28462.429,E2 28462.429} C_VEL
LIN {X 0,Y 586.6,Z 1031.549,A -85,B 0,C 180,E1 28461.548,E2 28461.548} C_VEL
LIN {X 0,Y 586.183,Z 1044.193,A -85,B 0,C 180,E1 28460.54,E2 28460.54} C_VEL
LIN {X 0,Y 585.776,Z 1056.347,A -85,B 0,C 180,E1 28459.336,E2 28459.336} C_VEL
LIN {X 0,Y 585.392,Z 1066.92,A -85,B 0,C 180,E1 28458.006,E2 28458.006} C_VEL
LIN {X 0,Y 585.119,Z 1075.307,A -85,B 0,C 180,E1 28456.681,E2 28456.681} C_VEL
LIN {X 0,Y 584.904,Z 1082.213,A -85,B 0,C 180,E1 28455.261,E2 28455.261} C_VEL
LIN {X 0,Y 584.774,Z 1087.665,A -85,B 0,C 180,E1 28453.747,E2 28453.747} C_VEL
LIN {X 0,Y 584.685,Z 1091.573,A -85,B 0,C 180,E1 28452.04,E2 28452.04} C_VEL
LIN {X 0,Y 584.673,Z 1093.313,A -85,B 0,C 180,E1 28450.484,E2 28450.484} C_VEL
LIN {X 0,Y 584.718,Z 1093.21,A -85,B 0,C 180,E1 28448.851,E2 28448.851} C_VEL
LIN {X 0,Y 584.81,Z 1091.3,A -85,B 0,C 180,E1 28447.266,E2 28447.266} C_VEL
LIN {X 0,Y 584.968,Z 1087.486,A -85,B 0,C 180,E1 28445.687,E2 28445.687} C_VEL
LIN {X 0,Y 585.193,Z 1082.11,A -85,B 0,C 180,E1 28444.211,E2 28444.211} C_VEL
LIN {X 0,Y 585.499,Z 1074.727,A -85,B 0,C 180,E1 28442.739,E2 28442.739} C_VEL
LIN {X 0,Y 585.854,Z 1066.494,A -85,B 0,C 180,E1 28441.465,E2 28441.465} C_VEL
LIN {X 0,Y 586.292,Z 1056.049,A -85,B 0,C 180,E1 28440.193,E2 28440.193} C_VEL
LIN {X 0,Y 586.745,Z 1044.548,A -85,B 0,C 180,E1 28439.07,E2 28439.07} C_VEL
LIN {X 0,Y 587.194,Z 1031.349,A -85,B 0,C 180,E1 28438.046,E2 28438.046} C_VEL
LIN {X 0,Y 587.548,Z 1017.939,A -85,B 0,C 180,E1 28437.218,E2 28437.218} C_VEL
LIN {X 0,Y 587.854,Z 1003.441,A -85,B 0,C 180,E1 28436.536,E2 28436.536} C_VEL
LIN {X 0,Y 588.065,Z 989.964,A -85,B 0,C 180,E1 28436.055,E2 28436.055} C_VEL
LIN {X 0,Y 588.175,Z 974.948,A -85,B 0,C 180,E1 28435.666,E2 28435.666} C_VEL
LIN {X 0,Y 588.408,Z 933.283,A -85,B 0,C 180,E1 28435.072,E2 28435.072} C_VEL
LIN {X 0,Y 589.798,Z 832.697,A -85,B 0,C 180,E1 28433.647,E2 28433.647} C_VEL
LIN {X 0,Y 590.663,Z 796.169,A -85,B 0,C 180,E1 28430.891,E2 28430.891} C_VEL
LIN {X 0,Y 591.358,Z 754.25,A -85,B 0,C 180,E1 28427.759,E2 28427.759} C_VEL
LIN {X 0,Y 591.922,Z 713.392,A -85,B 0,C 180,E1 28424.769,E2 28424.769} C_VEL
LIN {X 0,Y 592.193,Z 672.821,A -85,B 0,C 180,E1 28421.847,E2 28421.847} C_VEL
LIN {X 0,Y 592.211,Z 650.325,A -85,B 0,C 180,E1 28420.263,E2 28420.263} C_VEL
LIN {X 0,Y 587.021,Z 633.206,A -85,B 0,C 180,E1 28418.773,E2 28418.773} C_VEL
LIN {X 0,Y 585.262,Z 627.772,A -85,B 0,C 180,E1 28418.264,E2 28418.264} C_VEL
LIN {X 0,Y 585.224,Z 627.777,A -85,B 0,C 180,E1 28414.82,E2 28414.82} C_VEL
LIN {X 0,Y 585.262,Z 627.768,A -85,B 0,C 180,E1 28411.62,E2 28411.62} C_VEL
LIN {X 0,Y 585.235,Z 627.77,A -85,B 0,C 180,E1 28408.477,E2 28408.477} C_VEL
LIN {X 0,Y 585.254,Z 627.767,A -85,B 0,C 180,E1 28404.965,E2 28404.965} C_VEL
LIN {X 0,Y 585.265,Z 627.767,A -85,B 0,C 180,E1 28401.641,E2 28401.641} C_VEL
LIN {X 0,Y 585.219,Z 627.77,A -85,B 0,C 180,E1 28398.298,E2 28398.298} C_VEL
LIN {X 0,Y 585.259,Z 627.767,A -85,B 0,C 180,E1 28395.121,E2 28395.121} C_VEL
LIN {X 0,Y 585.244,Z 627.769,A -85,B 0,C 180,E1 28391.912,E2 28391.912} C_VEL
LIN {X 0,Y 585.265,Z 627.923,A -85,B 0,C 180,E1 28388.668,E2 28388.668} C_VEL
LIN {X 0,Y 593.428,Z 652.954,A -85,B 0,C 180,E1 28385.659,E2 28385.659} C_VEL
LIN {X 0,Y 597.77,Z 667.399,A -85,B 0,C 180,E1 28384.02,E2 28384.02} C_VEL
LIN {X 0,Y 597.042,Z 679.949,A -85,B 0,C 180,E1 28382.92,E2 28382.92} C_VEL
LIN {X 0,Y 604.073,Z 714.947,A -85,B 0,C 180,E1 28381.979,E2 28381.979} C_VEL
LIN {X 0,Y 599.485,Z 936.2,A -85,B 0,C 180,E1 28378.944,E2 28378.944} C_VEL
LIN {X 0,Y 598.475,Z 985.89,A -85,B 0,C 180,E1 28378.249,E2 28378.249} C_VEL
LIN {X 0,Y 597.596,Z 1007.559,A -85,B 0,C 180,E1 28377.782,E2 28377.782} C_VEL
LIN {X 0,Y 596.494,Z 1029.013,A -85,B 0,C 180,E1 28377.151,E2 28377.151} C_VEL
LIN {X 0,Y 595.282,Z 1049.737,A -85,B 0,C 180,E1 28376.375,E2 28376.375} C_VEL
LIN {X 0,Y 593.908,Z 1070.265,A -85,B 0,C 180,E1 28375.422,E2 28375.422} C_VEL
LIN {X 0,Y 592.473,Z 1089.938,A -85,B 0,C 180,E1 28374.315,E2 28374.315} C_VEL
LIN {X 0,Y 590.959,Z 1109.577,A -85,B 0,C 180,E1 28373.005,E2 28373.005} C_VEL
LIN {X 0,Y 589.667,Z 1126.558,A -85,B 0,C 180,E1 28371.681,E2 28371.681} C_VEL
LIN {X 0,Y 588.319,Z 1143.469,A -85,B 0,C 180,E1 28370.129,E2 28370.129} C_VEL
LIN {X 0,Y 587.144,Z 1159.098,A -85,B 0,C 180,E1 28368.455,E2 28368.455} C_VEL
LIN {X 0,Y 586.192,Z 1172.803,A -85,B 0,C 180,E1 28366.753,E2 28366.753} C_VEL
LIN {X 0,Y 585.41,Z 1185.197,A -85,B 0,C 180,E1 28364.944,E2 28364.944} C_VEL
LIN {X 0,Y 584.815,Z 1196.21,A -85,B 0,C 180,E1 28363.042,E2 28363.042} C_VEL
LIN {X 0,Y 584.391,Z 1205.88,A -85,B 0,C 180,E1 28361.046,E2 28361.046} C_VEL
LIN {X 0,Y 584.138,Z 1213.678,A -85,B 0,C 180,E1 28359.059,E2 28359.059} C_VEL
LIN {X 0,Y 583.993,Z 1220.007,A -85,B 0,C 180,E1 28356.981,E2 28356.981} C_VEL
LIN {X 0,Y 583.936,Z 1224.676,A -85,B 0,C 180,E1 28354.91,E2 28354.91} C_VEL
LIN {X 0,Y 583.929,Z 1227.521,A -85,B 0,C 180,E1 28352.943,E2 28352.943} C_VEL
LIN {X 0,Y 583.938,Z 1228.992,A -85,B 0,C 180,E1 28350.784,E2 28350.784} C_VEL
LIN {X 0,Y 583.929,Z 1228.83,A -85,B 0,C 180,E1 28348.723,E2 28348.723} C_VEL
LIN {X 0,Y 583.933,Z 1226.96,A -85,B 0,C 180,E1 28346.661,E2 28346.661} C_VEL
LIN {X 0,Y 583.958,Z 1223.326,A -85,B 0,C 180,E1 28344.496,E2 28344.496} C_VEL
LIN {X 0,Y 584.027,Z 1218.152,A -85,B 0,C 180,E1 28342.424,E2 28342.424} C_VEL
LIN {X 0,Y 584.192,Z 1211.141,A -85,B 0,C 180,E1 28340.361,E2 28340.361} C_VEL
LIN {X 0,Y 584.508,Z 1202.067,A -85,B 0,C 180,E1 28338.253,E2 28338.253} C_VEL
LIN {X 0,Y 584.953,Z 1192.107,A -85,B 0,C 180,E1 28336.355,E2 28336.355} C_VEL
LIN {X 0,Y 585.589,Z 1180.047,A -85,B 0,C 180,E1 28334.449,E2 28334.449} C_VEL
LIN {X 0,Y 586.391,Z 1166.454,A -85,B 0,C 180,E1 28332.637,E2 28332.637} C_VEL
LIN {X 0,Y 587.381,Z 1151.403,A -85,B 0,C 180,E1 28330.922,E2 28330.922} C_VEL
LIN {X 0,Y 588.493,Z 1135.367,A -85,B 0,C 180,E1 28329.355,E2 28329.355} C_VEL
LIN {X 0,Y 589.71,Z 1117.696,A -85,B 0,C 180,E1 28327.887,E2 28327.887} C_VEL
LIN {X 0,Y 591.032,Z 1098.402,A -85,B 0,C 180,E1 28326.52,E2 28326.52} C_VEL
LIN {X 0,Y 592.341,Z 1079.052,A -85,B 0,C 180,E1 28325.357,E2 28325.357} C_VEL
LIN {X 0,Y 593.645,Z 1058.194,A -85,B 0,C 180,E1 28324.307,E2 28324.307} C_VEL
LIN {X 0,Y 594.853,Z 1036.967,A -85,B 0,C 180,E1 28323.44,E2 28323.44} C_VEL
LIN {X 0,Y 595.988,Z 1014.145,A -85,B 0,C 180,E1 28322.696,E2 28322.696} C_VEL
LIN {X 0,Y 597.008,Z 991.095,A -85,B 0,C 180,E1 28322.134,E2 28322.134} C_VEL
LIN {X 0,Y 597.717,Z 967.654,A -85,B 0,C 180,E1 28321.736,E2 28321.736} C_VEL
LIN {X 0,Y 600.08,Z 857.845,A -85,B 0,C 180,E1 28320.159,E2 28320.159} C_VEL
LIN {X 0,Y 603.757,Z 748.843,A -85,B 0,C 180,E1 28318.433,E2 28318.433} C_VEL
LIN {X 0,Y 605.036,Z 713.496,A -85,B 0,C 180,E1 28317.822,E2 28317.822} C_VEL
LIN {X 0,Y 600.579,Z 685.904,A -85,B 0,C 180,E1 28316.893,E2 28316.893} C_VEL
LIN {X 0,Y 597.732,Z 671.62,A -85,B 0,C 180,E1 28316.313,E2 28316.313} C_VEL
LIN {X 0,Y 597.978,Z 666.753,A -85,B 0,C 180,E1 28315.817,E2 28315.817} C_VEL
LIN {X 0,Y 594.795,Z 654.08,A -85,B 0,C 180,E1 28314.124,E2 28314.124} C_VEL
LIN {X 0,Y 591.371,Z 643.611,A -85,B 0,C 180,E1 28312.467,E2 28312.467} C_VEL
LIN {X 0,Y 588.345,Z 635.339,A -85,B 0,C 180,E1 28310.911,E2 28310.911} C_VEL
LIN {X 0,Y 586.491,Z 631.167,A -85,B 0,C 180,E1 28309.952,E2 28309.952} C_VEL
LIN {X 0,Y 585.241,Z 627.771,A -85,B 0,C 180,E1 28309.088,E2 28309.088} C_VEL
LIN {X 0,Y 585.23,Z 627.773,A -85,B 0,C 180,E1 28305.717,E2 28305.717} C_VEL
LIN {X 0,Y 585.258,Z 627.768,A -85,B 0,C 180,E1 28302.576,E2 28302.576} C_VEL
LIN {X 0,Y 585.212,Z 627.774,A -85,B 0,C 180,E1 28299.44,E2 28299.44} C_VEL
LIN {X 0,Y 585.224,Z 627.856,A -85,B 0,C 180,E1 28297.069,E2 28297.069} C_VEL
LIN {X 0,Y 587.058,Z 632.797,A -85,B 0,C 180,E1 28295.749,E2 28295.749} C_VEL
LIN {X 0,Y 589.612,Z 638.884,A -85,B 0,C 180,E1 28294.369,E2 28294.369} C_VEL
LIN {X 0,Y 598.148,Z 651.987,A -85,B 0,C 180,E1 28293.188,E2 28293.188} C_VEL
LIN {X 0,Y 605.949,Z 666.106,A -85,B 0,C 180,E1 28292.212,E2 28292.212} C_VEL
LIN {X 0,Y 606.426,Z 667.737,A -85,B 0,C 180,E1 28292.141,E2 28292.141} C_VEL
LIN {X 0,Y 602.088,Z 771.709,A -85,B 0,C 180,E1 28290.409,E2 28290.409} C_VEL
LIN {X 0,Y 599.115,Z 875.646,A -85,B 0,C 180,E1 28288.83,E2 28288.83} C_VEL
LIN {X 0,Y 597.819,Z 935.614,A -85,B 0,C 180,E1 28287.951,E2 28287.951} C_VEL
LIN {X 0,Y 597.062,Z 958.771,A -85,B 0,C 180,E1 28287.428,E2 28287.428} C_VEL
LIN {X 0,Y 596.102,Z 980.054,A -85,B 0,C 180,E1 28286.77,E2 28286.77} C_VEL
LIN {X 0,Y 594.941,Z 1001.816,A -85,B 0,C 180,E1 28285.912,E2 28285.912} C_VEL
LIN {X 0,Y 593.739,Z 1021.628,A -85,B 0,C 180,E1 28284.954,E2 28284.954} C_VEL
LIN {X 0,Y 592.388,Z 1041.513,A -85,B 0,C 180,E1 28283.793,E2 28283.793} C_VEL
LIN {X 0,Y 591.038,Z 1059.618,A -85,B 0,C 180,E1 28282.526,E2 28282.526} C_VEL
LIN {X 0,Y 589.669,Z 1077.358,A -85,B 0,C 180,E1 28281.07,E2 28281.07} C_VEL
LIN {X 0,Y 588.439,Z 1093.105,A -85,B 0,C 180,E1 28279.559,E2 28279.559} C_VEL
LIN {X 0,Y 587.34,Z 1107.43,A -85,B 0,C 180,E1 28277.949,E2 28277.949} C_VEL
LIN {X 0,Y 586.37,Z 1120.401,A -85,B 0,C 180,E1 28276.242,E2 28276.242} C_VEL
LIN {X 0,Y 585.571,Z 1132.127,A -85,B 0,C 180,E1 28274.438,E2 28274.438} C_VEL
LIN {X 0,Y 584.96,Z 1142.451,A -85,B 0,C 180,E1 28272.54,E2 28272.54} C_VEL
LIN {X 0,Y 584.498,Z 1151.343,A -85,B 0,C 180,E1 28270.549,E2 28270.549} C_VEL
LIN {X 0,Y 584.213,Z 1158.528,A -85,B 0,C 180,E1 28268.565,E2 28268.565} C_VEL
LIN {X 0,Y 584.055,Z 1164.034,A -85,B 0,C 180,E1 28266.588,E2 28266.588} C_VEL
LIN {X 0,Y 583.978,Z 1168.176,A -85,B 0,C 180,E1 28264.519,E2 28264.519} C_VEL
LIN {X 0,Y 583.944,Z 1170.819,A -85,B 0,C 180,E1 28262.456,E2 28262.456} C_VEL
LIN {X 0,Y 583.933,Z 1171.817,A -85,B 0,C 180,E1 28260.395,E2 28260.395} C_VEL
LIN {X 0,Y 583.942,Z 1171.294,A -85,B 0,C 180,E1 28258.236,E2 28258.236} C_VEL
LIN {X 0,Y 583.954,Z 1169.287,A -85,B 0,C 180,E1 28256.173,E2 28256.173} C_VEL
LIN {X 0,Y 584.002,Z 1165.612,A -85,B 0,C 180,E1 28254.106,E2 28254.106} C_VEL
LIN {X 0,Y 584.14,Z 1160.083,A -85,B 0,C 180,E1 28251.934,E2 28251.934} C_VEL
LIN {X 0,Y 584.404,Z 1153.075,A -85,B 0,C 180,E1 28249.852,E2 28249.852} C_VEL
LIN {X 0,Y 584.801,Z 1144.525,A -85,B 0,C 180,E1 28247.862,E2 28247.862} C_VEL
LIN {X 0,Y 585.402,Z 1134.109,A -85,B 0,C 180,E1 28245.865,E2 28245.865} C_VEL
LIN {X 0,Y 586.206,Z 1122.261,A -85,B 0,C 180,E1 28243.962,E2 28243.962} C_VEL
LIN {X 0,Y 587.141,Z 1109.695,A -85,B 0,C 180,E1 28242.254,E2 28242.254} C_VEL
LIN {X 0,Y 588.294,Z 1094.961,A -85,B 0,C 180,E1 28240.544,E2 28240.544} C_VEL
LIN {X 0,Y 589.637,Z 1078.75,A -85,B 0,C 180,E1 28238.933,E2 28238.933} C_VEL
LIN {X 0,Y 591.054,Z 1061.53,A -85,B 0,C 180,E1 28237.47,E2 28237.47} C_VEL
LIN {X 0,Y 592.484,Z 1043.296,A -85,B 0,C 180,E1 28236.163,E2 28236.163} C_VEL
LIN {X 0,Y 593.898,Z 1024.268,A -85,B 0,C 180,E1 28235.005,E2 28235.005} C_VEL
LIN {X 0,Y 595.266,Z 1004.634,A -85,B 0,C 180,E1 28234,E2 28234} C_VEL
LIN {X 0,Y 596.483,Z 984.142,A -85,B 0,C 180,E1 28233.146,E2 28233.146} C_VEL
LIN {X 0,Y 597.583,Z 962.689,A -85,B 0,C 180,E1 28232.438,E2 28232.438} C_VEL
LIN {X 0,Y 598.448,Z 940.781,A -85,B 0,C 180,E1 28231.89,E2 28231.89} C_VEL
LIN {X 0,Y 599.103,Z 918.122,A -85,B 0,C 180,E1 28231.501,E2 28231.501} C_VEL
LIN {X 0,Y 603.468,Z 700.674,A -85,B 0,C 180,E1 28228.545,E2 28228.545} C_VEL
LIN {X 0,Y 604.168,Z 665.157,A -85,B 0,C 180,E1 28228.038,E2 28228.038} C_VEL
LIN {X 0,Y 591.141,Z 639.666,A -85,B 0,C 180,E1 28226.876,E2 28226.876} C_VEL
LIN {X 0,Y 586.314,Z 630.908,A -85,B 0,C 180,E1 28226.439,E2 28226.439} C_VEL
LIN {X 0,Y 585.251,Z 628.023,A -85,B 0,C 180,E1 28226.309,E2 28226.309} C_VEL
LIN {X 0,Y 585.203,Z 627.771,A -85,B 0,C 180,E1 28223.856,E2 28223.856} C_VEL
LIN {X 0,Y 584.215,Z 627.898,A -85,B 0,C 180,E1 28223.102,E2 28223.102} C_VEL
LIN {X 0,Y 577.845,Z 628.691,A -85,B 0,C 180,E1 28220.985,E2 28220.985} C_VEL
LIN {X 0,Y 577.323,Z 628.75,A -85,B 0,C 180,E1 28220.434,E2 28220.434} C_VEL
LIN {X 0,Y 577.306,Z 628.757,A -85,B 0,C 180,E1 28217.108,E2 28217.108} C_VEL
LIN {X 0,Y 577.317,Z 628.757,A -85,B 0,C 180,E1 28213.766,E2 28213.766} C_VEL
LIN {X 0,Y 577.256,Z 628.761,A -85,B 0,C 180,E1 28210.657,E2 28210.657} C_VEL
LIN {X 0,Y 577.251,Z 628.759,A -85,B 0,C 180,E1 28207.32,E2 28207.32} C_VEL
LIN {X 0,Y 577.323,Z 628.756,A -85,B 0,C 180,E1 28204.256,E2 28204.256} C_VEL
LIN {X 0,Y 577.314,Z 628.758,A -85,B 0,C 180,E1 28200.958,E2 28200.958} C_VEL
LIN {X 0,Y 577.324,Z 628.754,A -85,B 0,C 180,E1 28197.657,E2 28197.657} C_VEL
LIN {X 0,Y 577.262,Z 628.761,A -85,B 0,C 180,E1 28194.456,E2 28194.456} C_VEL
LIN {X 0,Y 577.267,Z 628.762,A -85,B 0,C 180,E1 28191.225,E2 28191.225} C_VEL
LIN {X 0,Y 577.281,Z 628.757,A -85,B 0,C 180,E1 28188.167,E2 28188.167} C_VEL
LIN {X 0,Y 577.29,Z 628.754,A -85,B 0,C 180,E1 28184.854,E2 28184.854} C_VEL
LIN {X 0,Y 577.306,Z 628.753,A -85,B 0,C 180,E1 28181.693,E2 28181.693} C_VEL
LIN {X 0,Y 577.289,Z 628.753,A -85,B 0,C 180,E1 28178.367,E2 28178.367} C_VEL
LIN {X 0,Y 577.301,Z 628.758,A -85,B 0,C 180,E1 28175.225,E2 28175.225} C_VEL
LIN {X 0,Y 577.241,Z 628.753,A -85,B 0,C 180,E1 28171.964,E2 28171.964} C_VEL
LIN {X 0,Y 577.295,Z 628.753,A -85,B 0,C 180,E1 28168.711,E2 28168.711} C_VEL
LIN {X 0,Y 577.314,Z 628.749,A -85,B 0,C 180,E1 28165.531,E2 28165.531} C_VEL
LIN {X 0,Y 577.32,Z 628.756,A -85,B 0,C 180,E1 28162.238,E2 28162.238} C_VEL
LIN {X 0,Y 577.278,Z 628.746,A -85,B 0,C 180,E1 28159.119,E2 28159.119} C_VEL
LIN {X 0,Y 577.241,Z 628.76,A -85,B 0,C 180,E1 28155.865,E2 28155.865} C_VEL
LIN {X 0,Y 577.312,Z 628.757,A -85,B 0,C 180,E1 28152.774,E2 28152.774} C_VEL
LIN {X 0,Y 577.289,Z 628.756,A -85,B 0,C 180,E1 28149.522,E2 28149.522} C_VEL
LIN {X 0,Y 577.318,Z 628.75,A -85,B 0,C 180,E1 28146.202,E2 28146.202} C_VEL
LIN {X 0,Y 577.286,Z 628.757,A -85,B 0,C 180,E1 28143.014,E2 28143.014} C_VEL
LIN {X 0,Y 577.298,Z 628.76,A -85,B 0,C 180,E1 28139.794,E2 28139.794} C_VEL
LIN {X 0,Y 577.252,Z 628.762,A -85,B 0,C 180,E1 28136.697,E2 28136.697} C_VEL
LIN {X 0,Y 577.274,Z 628.757,A -85,B 0,C 180,E1 28133.43,E2 28133.43} C_VEL
LIN {X 0,Y 577.318,Z 628.755,A -85,B 0,C 180,E1 28130.258,E2 28130.258} C_VEL
LIN {X 0,Y 577.315,Z 628.754,A -85,B 0,C 180,E1 28126.957,E2 28126.957} C_VEL
LIN {X 0,Y 577.321,Z 628.754,A -85,B 0,C 180,E1 28123.621,E2 28123.621} C_VEL
LIN {X 0,Y 577.287,Z 628.853,A -85,B 0,C 180,E1 28122.05,E2 28122.05} C_VEL
LIN {X 0,Y 584.606,Z 655.676,A -85,B 0,C 180,E1 28119.61,E2 28119.61} C_VEL
LIN {X 0,Y 583.648,Z 701.786,A -85,B 0,C 180,E1 28116.043,E2 28116.043} C_VEL
LIN {X 0,Y 582.784,Z 742.555,A -85,B 0,C 180,E1 28112.886,E2 28112.886} C_VEL
LIN {X 0,Y 581.815,Z 782.717,A -85,B 0,C 180,E1 28109.777,E2 28109.777} C_VEL
LIN {X 0,Y 580.937,Z 824.943,A -85,B 0,C 180,E1 28106.525,E2 28106.525} C_VEL
LIN {X 0,Y 580.926,Z 828.632,A -85,B 0,C 180,E1 28106.272,E2 28106.272} C_VEL
LIN {X 0,Y 581.218,Z 836.56,A -85,B 0,C 180,E1 28106.153,E2 28106.153} C_VEL
LIN {X 0,Y 579.888,Z 971.393,A -85,B 0,C 180,E1 28104.29,E2 28104.29} C_VEL
LIN {X 0,Y 579.738,Z 987.726,A -85,B 0,C 180,E1 28103.881,E2 28103.881} C_VEL
LIN {X 0,Y 579.483,Z 1002.943,A -85,B 0,C 180,E1 28103.325,E2 28103.325} C_VEL
LIN {X 0,Y 579.132,Z 1017.899,A -85,B 0,C 180,E1 28102.588,E2 28102.588} C_VEL
LIN {X 0,Y 578.725,Z 1032.7,A -85,B 0,C 180,E1 28101.645,E2 28101.645} C_VEL
LIN {X 0,Y 578.287,Z 1045.409,A -85,B 0,C 180,E1 28100.613,E2 28100.613} C_VEL
LIN {X 0,Y 577.868,Z 1057.443,A -85,B 0,C 180,E1 28099.401,E2 28099.401} C_VEL
LIN {X 0,Y 577.47,Z 1067.995,A -85,B 0,C 180,E1 28098.053,E2 28098.053} C_VEL
LIN {X 0,Y 577.177,Z 1076.568,A -85,B 0,C 180,E1 28096.671,E2 28096.671} C_VEL
LIN {X 0,Y 576.95,Z 1083.78,A -85,B 0,C 180,E1 28095.143,E2 28095.143} C_VEL
LIN {X 0,Y 576.82,Z 1088.971,A -85,B 0,C 180,E1 28093.633,E2 28093.633} C_VEL
LIN {X 0,Y 576.738,Z 1092.579,A -85,B 0,C 180,E1 28092.005,E2 28092.005} C_VEL
LIN {X 0,Y 576.73,Z 1094.259,A -85,B 0,C 180,E1 28090.486,E2 28090.486} C_VEL
LIN {X 0,Y 576.779,Z 1094.195,A -85,B 0,C 180,E1 28088.849,E2 28088.849} C_VEL
LIN {X 0,Y 576.88,Z 1092.378,A -85,B 0,C 180,E1 28087.267,E2 28087.267} C_VEL
LIN {X 0,Y 577.048,Z 1088.616,A -85,B 0,C 180,E1 28085.666,E2 28085.666} C_VEL
LIN {X 0,Y 577.292,Z 1083.309,A -85,B 0,C 180,E1 28084.169,E2 28084.169} C_VEL
LIN {X 0,Y 577.618,Z 1075.971,A -85,B 0,C 180,E1 28082.677,E2 28082.677} C_VEL
LIN {X 0,Y 578,Z 1067.819,A -85,B 0,C 180,E1 28081.386,E2 28081.386} C_VEL
LIN {X 0,Y 578.468,Z 1057.47,A -85,B 0,C 180,E1 28080.097,E2 28080.097} C_VEL
LIN {X 0,Y 578.952,Z 1046.091,A -85,B 0,C 180,E1 28078.959,E2 28078.959} C_VEL
LIN {X 0,Y 579.43,Z 1032.994,A -85,B 0,C 180,E1 28077.921,E2 28077.921} C_VEL
LIN {X 0,Y 579.826,Z 1018.835,A -85,B 0,C 180,E1 28077.032,E2 28077.032} C_VEL
LIN {X 0,Y 580.148,Z 1004.271,A -85,B 0,C 180,E1 28076.342,E2 28076.342} C_VEL
LIN {X 0,Y 580.364,Z 991.03,A -85,B 0,C 180,E1 28075.864,E2 28075.864} C_VEL
LIN {X 0,Y 580.477,Z 976.04,A -85,B 0,C 180,E1 28075.469,E2 28075.469} C_VEL
LIN {X 0,Y 580.754,Z 932.21,A -85,B 0,C 180,E1 28074.832,E2 28074.832} C_VEL
LIN {X 0,Y 582.267,Z 833.658,A -85,B 0,C 180,E1 28073.391,E2 28073.391} C_VEL
LIN {X 0,Y 583.118,Z 799.389,A -85,B 0,C 180,E1 28070.795,E2 28070.795} C_VEL
LIN {X 0,Y 583.822,Z 760.101,A -85,B 0,C 180,E1 28067.837,E2 28067.837} C_VEL
LIN {X 0,Y 584.503,Z 719.321,A -85,B 0,C 180,E1 28064.825,E2 28064.825} C_VEL
LIN {X 0,Y 584.851,Z 677.172,A -85,B 0,C 180,E1 28061.766,E2 28061.766} C_VEL
LIN {X 0,Y 584.995,Z 653.134,A -85,B 0,C 180,E1 28060.058,E2 28060.058} C_VEL
LIN {X 0,Y 580.045,Z 636.828,A -85,B 0,C 180,E1 28058.616,E2 28058.616} C_VEL
LIN {X 0,Y 577.328,Z 628.759,A -85,B 0,C 180,E1 28057.869,E2 28057.869} C_VEL
LIN {X 0,Y 577.309,Z 628.763,A -85,B 0,C 180,E1 28054.45,E2 28054.45} C_VEL
LIN {X 0,Y 577.288,Z 628.761,A -85,B 0,C 180,E1 28051.208,E2 28051.208} C_VEL
LIN {X 0,Y 577.292,Z 628.759,A -85,B 0,C 180,E1 28048.11,E2 28048.11} C_VEL
LIN {X 0,Y 577.317,Z 628.756,A -85,B 0,C 180,E1 28044.776,E2 28044.776} C_VEL
LIN {X 0,Y 577.322,Z 628.756,A -85,B 0,C 180,E1 28041.359,E2 28041.359} C_VEL
LIN {X 0,Y 577.288,Z 628.759,A -85,B 0,C 180,E1 28038.137,E2 28038.137} C_VEL
LIN {X 0,Y 577.309,Z 628.754,A -85,B 0,C 180,E1 28034.895,E2 28034.895} C_VEL
LIN {X 0,Y 577.303,Z 628.758,A -85,B 0,C 180,E1 28031.686,E2 28031.686} C_VEL
LIN {X 0,Y 577.349,Z 628.915,A -85,B 0,C 180,E1 28029.114,E2 28029.114} C_VEL
LIN {X 0,Y 585.812,Z 654.839,A -85,B 0,C 180,E1 28025.953,E2 28025.953} C_VEL
LIN {X 0,Y 590.386,Z 669.907,A -85,B 0,C 180,E1 28024.211,E2 28024.211} C_VEL
LIN {X 0,Y 589.81,Z 679.67,A -85,B 0,C 180,E1 28023.352,E2 28023.352} C_VEL
LIN {X 0,Y 597.129,Z 716.411,A -85,B 0,C 180,E1 28022.345,E2 28022.345} C_VEL
LIN {X 0,Y 592.196,Z 940.7,A -85,B 0,C 180,E1 28019.218,E2 28019.218} C_VEL
LIN {X 0,Y 591.177,Z 986.124,A -85,B 0,C 180,E1 28018.564,E2 28018.564} C_VEL
LIN {X 0,Y 590.244,Z 1007.988,A -85,B 0,C 180,E1 28018.083,E2 28018.083} C_VEL
LIN {X 0,Y 589.072,Z 1029.58,A -85,B 0,C 180,E1 28017.434,E2 28017.434} C_VEL
LIN {X 0,Y 587.692,Z 1051.714,A -85,B 0,C 180,E1 28016.579,E2 28016.579} C_VEL
LIN {X 0,Y 586.273,Z 1071.977,A -85,B 0,C 180,E1 28015.614,E2 28015.614} C_VEL
LIN {X 0,Y 584.786,Z 1091.336,A -85,B 0,C 180,E1 28014.494,E2 28014.494} C_VEL
LIN {X 0,Y 583.263,Z 1109.989,A -85,B 0,C 180,E1 28013.22,E2 28013.22} C_VEL
LIN {X 0,Y 581.816,Z 1127.877,A -85,B 0,C 180,E1 28011.788,E2 28011.788} C_VEL
LIN {X 0,Y 580.426,Z 1144.771,A -85,B 0,C 180,E1 28010.204,E2 28010.204} C_VEL
LIN {X 0,Y 579.213,Z 1160.081,A -85,B 0,C 180,E1 28008.518,E2 28008.518} C_VEL
LIN {X 0,Y 578.149,Z 1174.692,A -85,B 0,C 180,E1 28006.636,E2 28006.636} C_VEL
LIN {X 0,Y 577.385,Z 1186.559,A -85,B 0,C 180,E1 28004.849,E2 28004.849} C_VEL
LIN {X 0,Y 576.787,Z 1197.29,A -85,B 0,C 180,E1 28002.921,E2 28002.921} C_VEL
LIN {X 0,Y 576.372,Z 1206.661,A -85,B 0,C 180,E1 28000.898,E2 28000.898} C_VEL
LIN {X 0,Y 576.122,Z 1214.287,A -85,B 0,C 180,E1 27998.884,E2 27998.884} C_VEL
LIN {X 0,Y 575.985,Z 1220.345,A -85,B 0,C 180,E1 27996.79,E2 27996.79} C_VEL
LIN {X 0,Y 575.945,Z 1224.771,A -85,B 0,C 180,E1 27994.679,E2 27994.679} C_VEL
LIN {X 0,Y 575.944,Z 1227.586,A -85,B 0,C 180,E1 27992.586,E2 27992.586} C_VEL
LIN {X 0,Y 575.941,Z 1228.665,A -85,B 0,C 180,E1 27990.496,E2 27990.496} C_VEL
LIN {X 0,Y 575.947,Z 1228.16,A -85,B 0,C 180,E1 27988.307,E2 27988.307} C_VEL
LIN {X 0,Y 575.951,Z 1226.047,A -85,B 0,C 180,E1 27986.216,E2 27986.216} C_VEL
LIN {X 0,Y 575.968,Z 1222.21,A -85,B 0,C 180,E1 27984.12,E2 27984.12} C_VEL
LIN {X 0,Y 576.052,Z 1216.72,A -85,B 0,C 180,E1 27982.017,E2 27982.017} C_VEL
LIN {X 0,Y 576.234,Z 1209.763,A -85,B 0,C 180,E1 27980.006,E2 27980.006} C_VEL
LIN {X 0,Y 576.559,Z 1200.949,A -85,B 0,C 180,E1 27977.987,E2 27977.987} C_VEL
LIN {X 0,Y 577.062,Z 1190.184,A -85,B 0,C 180,E1 27975.96,E2 27975.96} C_VEL
LIN {X 0,Y 577.727,Z 1178.587,A -85,B 0,C 180,E1 27974.129,E2 27974.129} C_VEL
LIN {X 0,Y 578.532,Z 1165.581,A -85,B 0,C 180,E1 27972.394,E2 27972.394} C_VEL
LIN {X 0,Y 579.609,Z 1149.927,A -85,B 0,C 180,E1 27970.604,E2 27970.604} C_VEL
LIN {X 0,Y 580.791,Z 1133.708,A -85,B 0,C 180,E1 27969.016,E2 27969.016} C_VEL
LIN {X 0,Y 582.088,Z 1116.055,A -85,B 0,C 180,E1 27967.544,E2 27967.544} C_VEL
LIN {X 0,Y 583.451,Z 1097.084,A -85,B 0,C 180,E1 27966.196,E2 27966.196} C_VEL
LIN {X 0,Y 584.892,Z 1076.61,A -85,B 0,C 180,E1 27964.967,E2 27964.967} C_VEL
LIN {X 0,Y 586.242,Z 1056.351,A -85,B 0,C 180,E1 27963.947,E2 27963.947} C_VEL
LIN {X 0,Y 587.564,Z 1034.568,A -85,B 0,C 180,E1 27963.057,E2 27963.057} C_VEL
LIN {X 0,Y 588.725,Z 1012.216,A -85,B 0,C 180,E1 27962.332,E2 27962.332} C_VEL
LIN {X 0,Y 589.833,Z 988.287,A -85,B 0,C 180,E1 27961.755,E2 27961.755} C_VEL
LIN {X 0,Y 590.601,Z 962.902,A -85,B 0,C 180,E1 27961.333,E2 27961.333} C_VEL
LIN {X 0,Y 593.125,Z 859.102,A -85,B 0,C 180,E1 27959.79,E2 27959.79} C_VEL
LIN {X 0,Y 597.067,Z 753.212,A -85,B 0,C 180,E1 27958.059,E2 27958.059} C_VEL
LIN {X 0,Y 598.647,Z 715.036,A -85,B 0,C 180,E1 27957.378,E2 27957.378} C_VEL
LIN {X 0,Y 594.708,Z 689.088,A -85,B 0,C 180,E1 27956.471,E2 27956.471} C_VEL
LIN {X 0,Y 591.083,Z 670.599,A -85,B 0,C 180,E1 27955.685,E2 27955.685} C_VEL
LIN {X 0,Y 588.053,Z 658.057,A -85,B 0,C 180,E1 27953.961,E2 27953.961} C_VEL
LIN {X 0,Y 584.722,Z 647.609,A -85,B 0,C 180,E1 27952.251,E2 27952.251} C_VEL
LIN {X 0,Y 581.747,Z 639.65,A -85,B 0,C 180,E1 27950.666,E2 27950.666} C_VEL
LIN {X 0,Y 580.157,Z 635.921,A -85,B 0,C 180,E1 27949.776,E2 27949.776} C_VEL
LIN {X 0,Y 578.755,Z 632.425,A -85,B 0,C 180,E1 27948.833,E2 27948.833} C_VEL
LIN {X 0,Y 577.289,Z 628.762,A -85,B 0,C 180,E1 27947.641,E2 27947.641} C_VEL
LIN {X 0,Y 577.322,Z 628.758,A -85,B 0,C 180,E1 27944.405,E2 27944.405} C_VEL
LIN {X 0,Y 577.278,Z 628.763,A -85,B 0,C 180,E1 27941.164,E2 27941.164} C_VEL
LIN {X 0,Y 577.324,Z 628.794,A -85,B 0,C 180,E1 27938.574,E2 27938.574} C_VEL
LIN {X 0,Y 578.886,Z 632.673,A -85,B 0,C 180,E1 27937.224,E2 27937.224} C_VEL
LIN {X 0,Y 580.783,Z 637.738,A -85,B 0,C 180,E1 27935.817,E2 27935.817} C_VEL
LIN {X 0,Y 581.994,Z 640.434,A -85,B 0,C 180,E1 27935.178,E2 27935.178} C_VEL
LIN {X 0,Y 588.392,Z 649.736,A -85,B 0,C 180,E1 27934.191,E2 27934.191} C_VEL
LIN {X 0,Y 595.138,Z 660.704,A -85,B 0,C 180,E1 27933.251,E2 27933.251} C_VEL
LIN {X 0,Y 600.184,Z 670.305,A -85,B 0,C 180,E1 27932.59,E2 27932.59} C_VEL
LIN {X 0,Y 595.473,Z 771.06,A -85,B 0,C 180,E1 27930.85,E2 27930.85} C_VEL
LIN {X 0,Y 592.217,Z 871.111,A -85,B 0,C 180,E1 27929.27,E2 27929.27} C_VEL
LIN {X 0,Y 590.635,Z 936.435,A -85,B 0,C 180,E1 27928.283,E2 27928.283} C_VEL
LIN {X 0,Y 589.826,Z 959.519,A -85,B 0,C 180,E1 27927.75,E2 27927.75} C_VEL
LIN {X 0,Y 588.799,Z 980.94,A -85,B 0,C 180,E1 27927.074,E2 27927.074} C_VEL
LIN {X 0,Y 587.577,Z 1002.549,A -85,B 0,C 180,E1 27926.207,E2 27926.207} C_VEL
LIN {X 0,Y 586.31,Z 1022.276,A -85,B 0,C 180,E1 27925.238,E2 27925.238} C_VEL
LIN {X 0,Y 584.894,Z 1042.031,A -85,B 0,C 180,E1 27924.069,E2 27924.069} C_VEL
LIN {X 0,Y 583.471,Z 1060.163,A -85,B 0,C 180,E1 27922.784,E2 27922.784} C_VEL
LIN {X 0,Y 582.023,Z 1077.905,A -85,B 0,C 180,E1 27921.308,E2 27921.308} C_VEL
LIN {X 0,Y 580.774,Z 1093.174,A -85,B 0,C 180,E1 27919.828,E2 27919.828} C_VEL
LIN {X 0,Y 579.598,Z 1107.528,A -85,B 0,C 180,E1 27918.197,E2 27918.197} C_VEL
LIN {X 0,Y 578.543,Z 1120.882,A -85,B 0,C 180,E1 27916.422,E2 27916.422} C_VEL
LIN {X 0,Y 577.718,Z 1132.349,A -85,B 0,C 180,E1 27914.639,E2 27914.639} C_VEL
LIN {X 0,Y 577.055,Z 1142.794,A -85,B 0,C 180,E1 27912.698,E2 27912.698} C_VEL
LIN {X 0,Y 576.561,Z 1151.653,A -85,B 0,C 180,E1 27910.696,E2 27910.696} C_VEL
LIN {X 0,Y 576.252,Z 1158.875,A -85,B 0,C 180,E1 27908.684,E2 27908.684} C_VEL
LIN {X 0,Y 576.079,Z 1164.401,A -85,B 0,C 180,E1 27906.68,E2 27906.68} C_VEL
LIN {X 0,Y 575.994,Z 1168.564,A -85,B 0,C 180,E1 27904.582,E2 27904.582} C_VEL
LIN {X 0,Y 575.957,Z 1171.217,A -85,B 0,C 180,E1 27902.49,E2 27902.49} C_VEL
LIN {X 0,Y 575.944,Z 1172.211,A -85,B 0,C 180,E1 27900.4,E2 27900.4} C_VEL
LIN {X 0,Y 575.952,Z 1171.674,A -85,B 0,C 180,E1 27898.211,E2 27898.211} C_VEL
LIN {X 0,Y 575.965,Z 1169.652,A -85,B 0,C 180,E1 27896.12,E2 27896.12} C_VEL
LIN {X 0,Y 576.019,Z 1165.951,A -85,B 0,C 180,E1 27894.024,E2 27894.024} C_VEL
LIN {X 0,Y 576.173,Z 1160.379,A -85,B 0,C 180,E1 27891.821,E2 27891.821} C_VEL
LIN {X 0,Y 576.455,Z 1153.323,A -85,B 0,C 180,E1 27889.711,E2 27889.711} C_VEL
LIN {X 0,Y 576.882,Z 1144.732,A -85,B 0,C 180,E1 27887.693,E2 27887.693} C_VEL
LIN {X 0,Y 577.526,Z 1134.257,A -85,B 0,C 180,E1 27885.668,E2 27885.668} C_VEL
LIN {X 0,Y 578.384,Z 1122.341,A -85,B 0,C 180,E1 27883.739,E2 27883.739} C_VEL
LIN {X 0,Y 579.45,Z 1108.94,A -85,B 0,C 180,E1 27881.907,E2 27881.907} C_VEL
LIN {X 0,Y 580.601,Z 1094.888,A -85,B 0,C 180,E1 27880.275,E2 27880.275} C_VEL
LIN {X 0,Y 582.045,Z 1078.164,A -85,B 0,C 180,E1 27878.608,E2 27878.608} C_VEL
LIN {X 0,Y 583.51,Z 1061.266,A -85,B 0,C 180,E1 27877.165,E2 27877.165} C_VEL
LIN {X 0,Y 585.017,Z 1042.909,A -85,B 0,C 180,E1 27875.839,E2 27875.839} C_VEL
LIN {X 0,Y 586.506,Z 1023.695,A -85,B 0,C 180,E1 27874.668,E2 27874.668} C_VEL
LIN {X 0,Y 587.928,Z 1003.796,A -85,B 0,C 180,E1 27873.651,E2 27873.651} C_VEL
LIN {X 0,Y 589.255,Z 982.643,A -85,B 0,C 180,E1 27872.769,E2 27872.769} C_VEL
LIN {X 0,Y 590.362,Z 961.198,A -85,B 0,C 180,E1 27872.071,E2 27872.071} C_VEL
LIN {X 0,Y 591.263,Z 938.36,A -85,B 0,C 180,E1 27871.514,E2 27871.514} C_VEL
LIN {X 0,Y 591.94,Z 914.75,A -85,B 0,C 180,E1 27871.123,E2 27871.123} C_VEL
LIN {X 0,Y 596.307,Z 710.649,A -85,B 0,C 180,E1 27868.298,E2 27868.298} C_VEL
LIN {X 0,Y 597.226,Z 667.627,A -85,B 0,C 180,E1 27867.68,E2 27867.68} C_VEL
LIN {X 0,Y 583.169,Z 640.209,A -85,B 0,C 180,E1 27866.394,E2 27866.394} C_VEL
LIN {X 0,Y 578.431,Z 632.059,A -85,B 0,C 180,E1 27865.962,E2 27865.962} C_VEL
LIN {X 0,Y 577.245,Z 628.767,A -85,B 0,C 180,E1 27865.809,E2 27865.809} C_VEL
LIN {X 0,Y 577.325,Z 628.754,A -85,B 0,C 180,E1 27862.652,E2 27862.652} C_VEL
LIN {X 0,Y 577.323,Z 628.75,A -85,B 0,C 180,E1 27860.434,E2 27860.434} C_VEL
LIN {X 0,Y 576.339,Z 628.875,A -85,B 0,C 180,E1 27859.669,E2 27859.669} C_VEL
LIN {X 0,Y 569.903,Z 629.682,A -85,B 0,C 180,E1 27857.524,E2 27857.524} C_VEL
LIN {X 0,Y 569.363,Z 629.745,A -85,B 0,C 180,E1 27856.965,E2 27856.965} C_VEL
LIN {X 0,Y 569.368,Z 629.749,A -85,B 0,C 180,E1 27853.644,E2 27853.644} C_VEL
LIN {X 0,Y 569.326,Z 629.75,A -85,B 0,C 180,E1 27850.529,E2 27850.529} C_VEL
LIN {X 0,Y 569.312,Z 629.748,A -85,B 0,C 180,E1 27847.292,E2 27847.292} C_VEL
LIN {X 0,Y 569.384,Z 629.744,A -85,B 0,C 180,E1 27844.192,E2 27844.192} C_VEL
LIN {X 0,Y 569.383,Z 629.748,A -85,B 0,C 180,E1 27840.832,E2 27840.832} C_VEL
LIN {X 0,Y 569.386,Z 629.744,A -85,B 0,C 180,E1 27837.508,E2 27837.508} C_VEL
LIN {X 0,Y 569.326,Z 629.749,A -85,B 0,C 180,E1 27834.294,E2 27834.294} C_VEL
LIN {X 0,Y 569.303,Z 629.751,A -85,B 0,C 180,E1 27830.882,E2 27830.882} C_VEL
LIN {X 0,Y 569.378,Z 629.742,A -85,B 0,C 180,E1 27827.793,E2 27827.793} C_VEL
LIN {X 0,Y 569.357,Z 629.745,A -85,B 0,C 180,E1 27824.546,E2 27824.546} C_VEL
LIN {X 0,Y 569.379,Z 629.74,A -85,B 0,C 180,E1 27821.242,E2 27821.242} C_VEL
LIN {X 0,Y 569.335,Z 629.741,A -85,B 0,C 180,E1 27817.976,E2 27817.976} C_VEL
LIN {X 0,Y 569.351,Z 629.748,A -85,B 0,C 180,E1 27814.837,E2 27814.837} C_VEL
LIN {X 0,Y 569.326,Z 629.742,A -85,B 0,C 180,E1 27811.612,E2 27811.612} C_VEL
LIN {X 0,Y 569.339,Z 629.744,A -85,B 0,C 180,E1 27808.391,E2 27808.391} C_VEL
LIN {X 0,Y 569.374,Z 629.736,A -85,B 0,C 180,E1 27805.166,E2 27805.166} C_VEL
LIN {X 0,Y 569.364,Z 629.745,A -85,B 0,C 180,E1 27801.824,E2 27801.824} C_VEL
LIN {X 0,Y 569.379,Z 629.732,A -85,B 0,C 180,E1 27798.556,E2 27798.556} C_VEL
LIN {X 0,Y 569.298,Z 629.749,A -85,B 0,C 180,E1 27795.396,E2 27795.396} C_VEL
LIN {X 0,Y 569.334,Z 629.745,A -85,B 0,C 180,E1 27791.997,E2 27791.997} C_VEL
LIN {X 0,Y 569.381,Z 629.744,A -85,B 0,C 180,E1 27788.794,E2 27788.794} C_VEL
LIN {X 0,Y 569.378,Z 629.747,A -85,B 0,C 180,E1 27785.451,E2 27785.451} C_VEL
LIN {X 0,Y 569.383,Z 629.742,A -85,B 0,C 180,E1 27782.155,E2 27782.155} C_VEL
LIN {X 0,Y 569.305,Z 629.75,A -85,B 0,C 180,E1 27779.031,E2 27779.031} C_VEL
LIN {X 0,Y 569.342,Z 629.749,A -85,B 0,C 180,E1 27775.804,E2 27775.804} C_VEL
LIN {X 0,Y 569.368,Z 629.748,A -85,B 0,C 180,E1 27772.585,E2 27772.585} C_VEL
LIN {X 0,Y 569.365,Z 629.744,A -85,B 0,C 180,E1 27769.341,E2 27769.341} C_VEL
LIN {X 0,Y 569.364,Z 629.743,A -85,B 0,C 180,E1 27766.052,E2 27766.052} C_VEL
LIN {X 0,Y 569.328,Z 629.753,A -85,B 0,C 180,E1 27762.77,E2 27762.77} C_VEL
LIN {X 0,Y 569.352,Z 629.961,A -85,B 0,C 180,E1 27762.327,E2 27762.327} C_VEL
LIN {X 0,Y 576.823,Z 657.11,A -85,B 0,C 180,E1 27759.836,E2 27759.836} C_VEL
LIN {X 0,Y 576.445,Z 682.925,A -85,B 0,C 180,E1 27757.816,E2 27757.816} C_VEL
LIN {X 0,Y 575.548,Z 724.579,A -85,B 0,C 180,E1 27754.57,E2 27754.57} C_VEL
LIN {X 0,Y 574.605,Z 766.077,A -85,B 0,C 180,E1 27751.349,E2 27751.349} C_VEL
LIN {X 0,Y 573.521,Z 809.573,A -85,B 0,C 180,E1 27747.965,E2 27747.965} C_VEL
LIN {X 0,Y 573.177,Z 829.257,A -85,B 0,C 180,E1 27746.469,E2 27746.469} C_VEL
LIN {X 0,Y 573.474,Z 836.991,A -85,B 0,C 180,E1 27746.349,E2 27746.349} C_VEL
LIN {X 0,Y 572.066,Z 972.413,A -85,B 0,C 180,E1 27744.442,E2 27744.442} C_VEL
LIN {X 0,Y 571.911,Z 988.803,A -85,B 0,C 180,E1 27744.023,E2 27744.023} C_VEL
LIN {X 0,Y 571.639,Z 1004.294,A -85,B 0,C 180,E1 27743.446,E2 27743.446} C_VEL
LIN {X 0,Y 571.277,Z 1019.029,A -85,B 0,C 180,E1 27742.704,E2 27742.704} C_VEL
LIN {X 0,Y 570.873,Z 1033.146,A -85,B 0,C 180,E1 27741.794,E2 27741.794} C_VEL
LIN {X 0,Y 570.412,Z 1046.116,A -85,B 0,C 180,E1 27740.735,E2 27740.735} C_VEL
LIN {X 0,Y 569.995,Z 1057.602,A -85,B 0,C 180,E1 27739.573,E2 27739.573} C_VEL
LIN {X 0,Y 569.59,Z 1067.985,A -85,B 0,C 180,E1 27738.257,E2 27738.257} C_VEL
LIN {X 0,Y 569.268,Z 1076.992,A -85,B 0,C 180,E1 27736.819,E2 27736.819} C_VEL
LIN {X 0,Y 569.022,Z 1084.311,A -85,B 0,C 180,E1 27735.276,E2 27735.276} C_VEL
LIN {X 0,Y 568.883,Z 1089.717,A -85,B 0,C 180,E1 27733.724,E2 27733.724} C_VEL
LIN {X 0,Y 568.792,Z 1093.586,A -85,B 0,C 180,E1 27731.97,E2 27731.97} C_VEL
LIN {X 0,Y 568.785,Z 1095.225,A -85,B 0,C 180,E1 27730.43,E2 27730.43} C_VEL
LIN {X 0,Y 568.843,Z 1095.15,A -85,B 0,C 180,E1 27728.794,E2 27728.794} C_VEL
LIN {X 0,Y 568.955,Z 1093.265,A -85,B 0,C 180,E1 27727.165,E2 27727.165} C_VEL
LIN {X 0,Y 569.147,Z 1089.47,A -85,B 0,C 180,E1 27725.543,E2 27725.543} C_VEL
LIN {X 0,Y 569.415,Z 1084.103,A -85,B 0,C 180,E1 27724.025,E2 27724.025} C_VEL
LIN {X 0,Y 569.774,Z 1076.726,A -85,B 0,C 180,E1 27722.512,E2 27722.512} C_VEL
LIN {X 0,Y 570.187,Z 1068.483,A -85,B 0,C 180,E1 27721.204,E2 27721.204} C_VEL
LIN {X 0,Y 570.693,Z 1058.03,A -85,B 0,C 180,E1 27719.897,E2 27719.897} C_VEL
LIN {X 0,Y 571.208,Z 1046.503,A -85,B 0,C 180,E1 27718.744,E2 27718.744} C_VEL
LIN {X 0,Y 571.714,Z 1033.243,A -85,B 0,C 180,E1 27717.693,E2 27717.693} C_VEL
LIN {X 0,Y 572.11,Z 1019.73,A -85,B 0,C 180,E1 27716.842,E2 27716.842} C_VEL
LIN {X 0,Y 572.448,Z 1005.107,A -85,B 0,C 180,E1 27716.142,E2 27716.142} C_VEL
LIN {X 0,Y 572.677,Z 991.973,A -85,B 0,C 180,E1 27715.661,E2 27715.661} C_VEL
LIN {X 0,Y 572.8,Z 977.029,A -85,B 0,C 180,E1 27715.261,E2 27715.261} C_VEL
LIN {X 0,Y 573.098,Z 933.71,A -85,B 0,C 180,E1 27714.615,E2 27714.615} C_VEL
LIN {X 0,Y 574.755,Z 834.71,A -85,B 0,C 180,E1 27713.129,E2 27713.129} C_VEL
LIN {X 0,Y 575.734,Z 797.645,A -85,B 0,C 180,E1 27710.3,E2 27710.3} C_VEL
LIN {X 0,Y 576.497,Z 757.516,A -85,B 0,C 180,E1 27707.273,E2 27707.273} C_VEL
LIN {X 0,Y 577.192,Z 717.707,A -85,B 0,C 180,E1 27704.319,E2 27704.319} C_VEL
LIN {X 0,Y 577.628,Z 675.912,A -85,B 0,C 180,E1 27701.268,E2 27701.268} C_VEL
LIN {X 0,Y 577.827,Z 656.078,A -85,B 0,C 180,E1 27699.856,E2 27699.856} C_VEL
LIN {X 0,Y 573.041,Z 640.292,A -85,B 0,C 180,E1 27698.432,E2 27698.432} C_VEL
LIN {X 0,Y 569.38,Z 629.752,A -85,B 0,C 180,E1 27697.435,E2 27697.435} C_VEL
LIN {X 0,Y 569.386,Z 629.747,A -85,B 0,C 180,E1 27694.037,E2 27694.037} C_VEL
LIN {X 0,Y 569.346,Z 629.75,A -85,B 0,C 180,E1 27690.659,E2 27690.659} C_VEL
LIN {X 0,Y 569.375,Z 629.747,A -85,B 0,C 180,E1 27687.447,E2 27687.447} C_VEL
LIN {X 0,Y 569.356,Z 629.748,A -85,B 0,C 180,E1 27684.209,E2 27684.209} C_VEL
LIN {X 0,Y 569.377,Z 629.746,A -85,B 0,C 180,E1 27680.751,E2 27680.751} C_VEL
